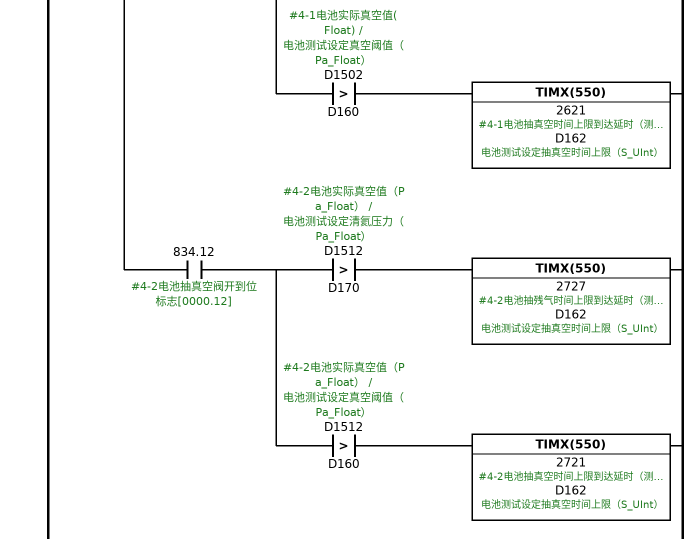
; [picture p648: Common / 动作延时, rungs 17-17]
; rung 17
LD P_On
OUT TR0
AND<=F(332) D1502 D160  ; #4-1电池实际真空值(Float), 电池测试设定真空阈值（Pa_Float）
LD 834.10  ; #4-1电池抽真空阀开到位标志[0000.10]
OR P_On
ANDLD
TIMX(550) 2620 #1  ; #4-1电池抽真空阈值到达延时（测试）
LD TR0
AND<=F(332) D1512 D160  ; #4-2电池实际真空值（Pa_Float）, 电池测试设定真空阈值（Pa_Float）
LD 834.12  ; #4-2电池抽真空阀开到位标志[0000.12]
OR P_On
ANDLD
TIMX(550) 2720 #1  ; #4-2电池抽真空阈值到达延时（测试）
LD TR0
LD>F(333) D1502 D172  ; #4-1电池实际真空值(Float), 电池测试设定破真空阈值（Pa_Float）
OR H5.15  ; 腔体模式（0-正压 1-负压）
ANDLD
TIMX(550) 2622 #1  ; #4-1电池破真空阈值到达延时（测试）
LD TR0
LD>F(333) D1512 D172  ; #4-2电池实际真空值（Pa_Float）, 电池测试设定破真空阈值（Pa_Float）
OR H5.15  ; 腔体模式（0-正压 1-负压）
ANDLD
TIMX(550) 2722 #1  ; #4-2电池破真空阈值到达延时（测试）
LD TR0
AND>=F(334) D1502 D176  ; #4-1电池实际真空值(Float), 电池测试设定注氦压力（Pa_Float）
AND 834.14  ; #4-1电池注氦阀开到位标志[0000.14]
TIMHX(551) 2624 #0  ; #4-1电池注氦压力到达延时（测试）
LD TR0
AND>=F(334) D1512 D176  ; #4-2电池实际真空值（Pa_Float）, 电池测试设定注氦压力（Pa_Float）
AND 835.00  ; #4-2电池注氦阀开到位标志[0000.00]
TIMHX(551) 2724 #0  ; #4-2电池注氦压力到达延时（测试）
LD TR0
AND<=F(332) D1502 D172  ; #4-1电池实际真空值(Float), 电池测试设定破真空阈值（Pa_Float）
AND 835.02  ; #4-1电池破真空阀开到位标志[0000.02]
TIMX(550) 2623 &20  ; #4-1电池破真空时间上限到达延时（测试）
LD TR0
AND<=F(332) D1512 D172  ; #4-2电池实际真空值（Pa_Float）, 电池测试设定破真空阈值（Pa_Float）
AND 835.04  ; #4-2电池破真空阀开到位标志[0000.04]
TIMX(550) 2723 &20  ; #4-2电池破真空时间上限到达延时（测试）
LD TR0
AND<=F(332) D1502 D170  ; #4-1电池实际真空值(Float), 电池测试设定清氦压力（Pa_Float）
TIMX(550) 2626 #1  ; #4-1电池抽残气压力到达延时（测试）
LD TR0
AND<=F(332) D1512 D170  ; #4-2电池实际真空值（Pa_Float）, 电池测试设定清氦压力（Pa_Float）
TIMX(550) 2726 #1  ; #4-2电池抽残气压力到达延时（测试）
LD TR0
AND>=F(334) D1502 D174  ; #4-1电池实际真空值(Float), 电池测试设定预抽检测压力（Pa_Float）
AND T2609  ; #4-1腔体预抽时间到达延时（测试）
TIMHX(551) 2628 #0  ; #4-1电池预抽压力正常判定延时（测试）
LD TR0
AND>=F(334) D1512 D174  ; #4-2电池实际真空值（Pa_Float）, 电池测试设定预抽检测压力（Pa_Float）
AND T2609  ; #4-1腔体预抽时间到达延时（测试）
TIMHX(551) 2728 #0  ; #4-2电池预抽压力正常判定延时（测试）
LD TR0
AND 834.14  ; #4-1电池注氦阀开到位标志[0000.14]
AND<F(331) D1502 D176  ; #4-1电池实际真空值(Float), 电池测试设定注氦压力（Pa_Float）
TIMX(550) 2625 D168  ; 电池测试设定注氦时间上限（S_UInt）, #4-1电池注氦时间上限到达延时（测试）
LD TR0
AND 835.00  ; #4-2电池注氦阀开到位标志[0000.00]
AND<F(331) D1512 D178  ; #4-2电池实际真空值（Pa_Float）, 注氦压力下限值（Pa_Float）
TIMX(550) 2725 D168  ; 电池测试设定注氦时间上限（S_UInt）, #4-2电池注氦时间上限到达延时（测试）
LD TR0
AND 834.10  ; #4-1电池抽真空阀开到位标志[0000.10]
OUT TR1
AND>F(333) D1502 D170  ; #4-1电池实际真空值(Float), 电池测试设定清氦压力（Pa_Float）
TIMX(550) 2627 D162  ; 电池测试设定抽真空时间上限（S_UInt）, #4-1电池抽残气时间上限到达延时（测试）
LD TR1
AND>F(333) D1502 D160  ; #4-1电池实际真空值(Float), 电池测试设定真空阈值（Pa_Float）
TIMX(550) 2621 D162  ; 电池测试设定抽真空时间上限（S_UInt）, #4-1电池抽真空时间上限到达延时（测试）
LD TR0
AND 834.12  ; #4-2电池抽真空阀开到位标志[0000.12]
OUT TR0
AND>F(333) D1512 D170  ; #4-2电池实际真空值（Pa_Float）, 电池测试设定清氦压力（Pa_Float）
TIMX(550) 2727 D162  ; 电池测试设定抽真空时间上限（S_UInt）, #4-2电池抽残气时间上限到达延时（测试）
LD TR0
AND>F(333) D1512 D160  ; #4-2电池实际真空值（Pa_Float）, 电池测试设定真空阈值（Pa_Float）
TIMX(550) 2721 D162  ; 电池测试设定抽真空时间上限（S_UInt）, #4-2电池抽真空时间上限到达延时（测试）

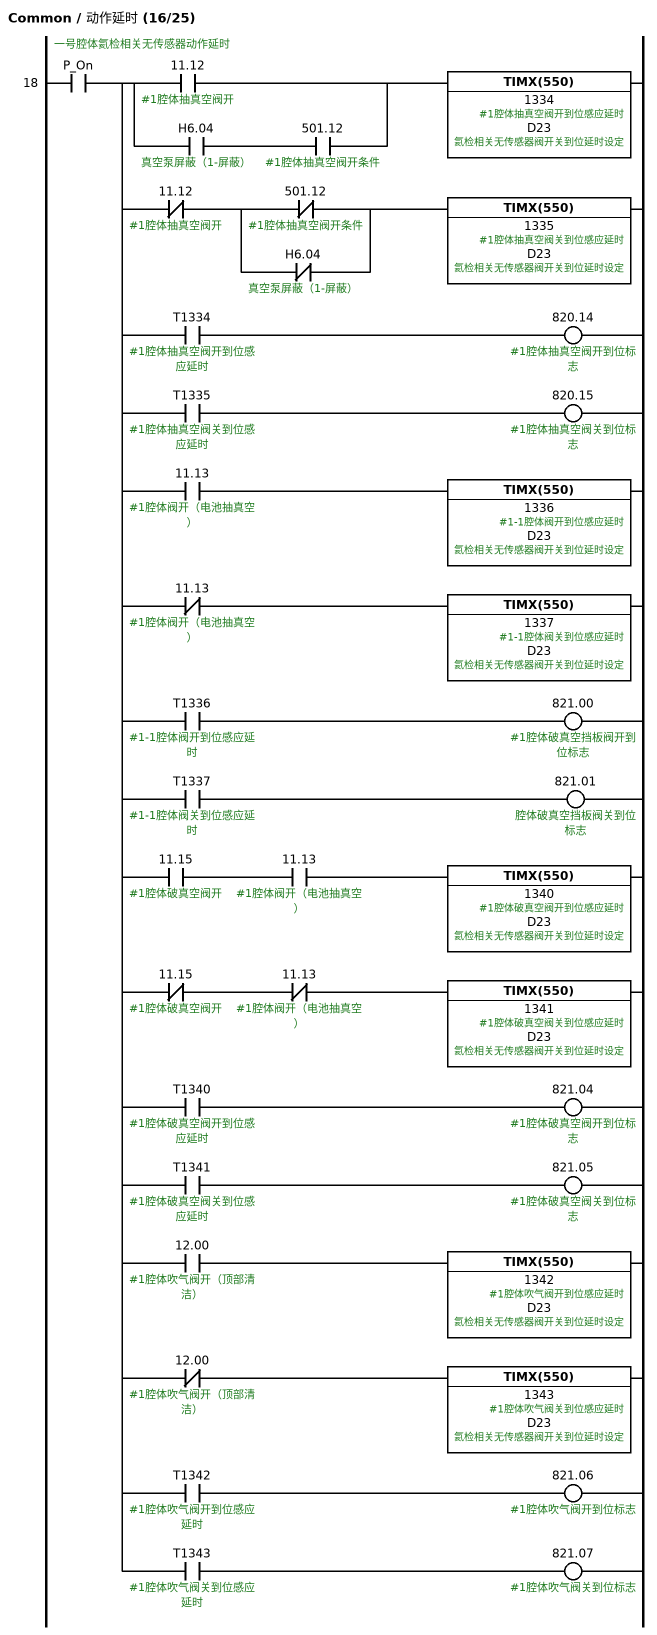
; rung 18: 一号腔体氦检相关无传感器动作延时
LD P_On
OUT TR0
LD 11.12  ; #1腔体抽真空阀开
LD H6.04  ; 真空泵屏蔽（1-屏蔽）
AND 501.12  ; #1腔体抽真空阀开条件
ORLD
ANDLD
TIMX(550) 1334 D23  ; 氦检相关无传感器阀开关到位延时设定, #1腔体抽真空阀开到位感应延时
LD TR0
ANDNOT 11.12  ; #1腔体抽真空阀开
LDNOT 501.12  ; #1腔体抽真空阀开条件
ORNOT H6.04  ; 真空泵屏蔽（1-屏蔽）
ANDLD
TIMX(550) 1335 D23  ; 氦检相关无传感器阀开关到位延时设定, #1腔体抽真空阀关到位感应延时
LD TR0
AND T1334  ; #1腔体抽真空阀开到位感应延时
OUT 820.14  ; #1腔体抽真空阀开到位标志
LD TR0
AND T1335  ; #1腔体抽真空阀关到位感应延时
OUT 820.15  ; #1腔体抽真空阀关到位标志
LD TR0
AND 11.13  ; #1腔体阀开（电池抽真空）
TIMX(550) 1336 D23  ; 氦检相关无传感器阀开关到位延时设定, #1-1腔体阀开到位感应延时
LD TR0
ANDNOT 11.13  ; #1腔体阀开（电池抽真空）
TIMX(550) 1337 D23  ; 氦检相关无传感器阀开关到位延时设定, #1-1腔体阀关到位感应延时
LD TR0
AND T1336  ; #1-1腔体阀开到位感应延时
OUT 821.00  ; #1腔体破真空挡板阀开到位标志
LD TR0
AND T1337  ; #1-1腔体阀关到位感应延时
OUT 821.01  ; 腔体破真空挡板阀关到位标志
LD TR0
AND 11.15  ; #1腔体破真空阀开
AND 11.13  ; #1腔体阀开（电池抽真空）
TIMX(550) 1340 D23  ; 氦检相关无传感器阀开关到位延时设定, #1腔体破真空阀开到位感应延时
LD TR0
ANDNOT 11.15  ; #1腔体破真空阀开
ANDNOT 11.13  ; #1腔体阀开（电池抽真空）
TIMX(550) 1341 D23  ; 氦检相关无传感器阀开关到位延时设定, #1腔体破真空阀关到位感应延时
LD TR0
AND T1340  ; #1腔体破真空阀开到位感应延时
OUT 821.04  ; #1腔体破真空阀开到位标志
LD TR0
AND T1341  ; #1腔体破真空阀关到位感应延时
OUT 821.05  ; #1腔体破真空阀关到位标志
LD TR0
AND 12.00  ; #1腔体吹气阀开（顶部清洁）
TIMX(550) 1342 D23  ; 氦检相关无传感器阀开关到位延时设定, #1腔体吹气阀开到位感应延时
LD TR0
ANDNOT 12.00  ; #1腔体吹气阀开（顶部清洁）
TIMX(550) 1343 D23  ; 氦检相关无传感器阀开关到位延时设定, #1腔体吹气阀关到位感应延时
LD TR0
AND T1342  ; #1腔体吹气阀开到位感应延时
OUT 821.06  ; #1腔体吹气阀开到位标志
LD TR0
AND T1343  ; #1腔体吹气阀关到位感应延时
OUT 821.07  ; #1腔体吹气阀关到位标志

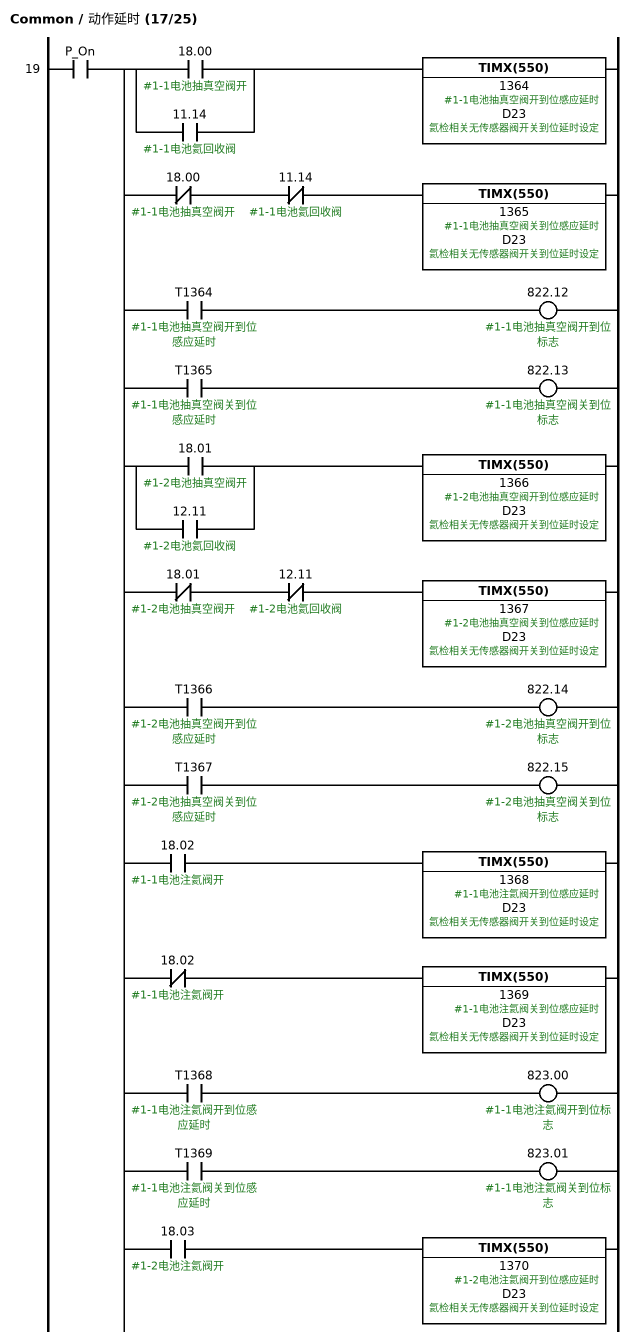

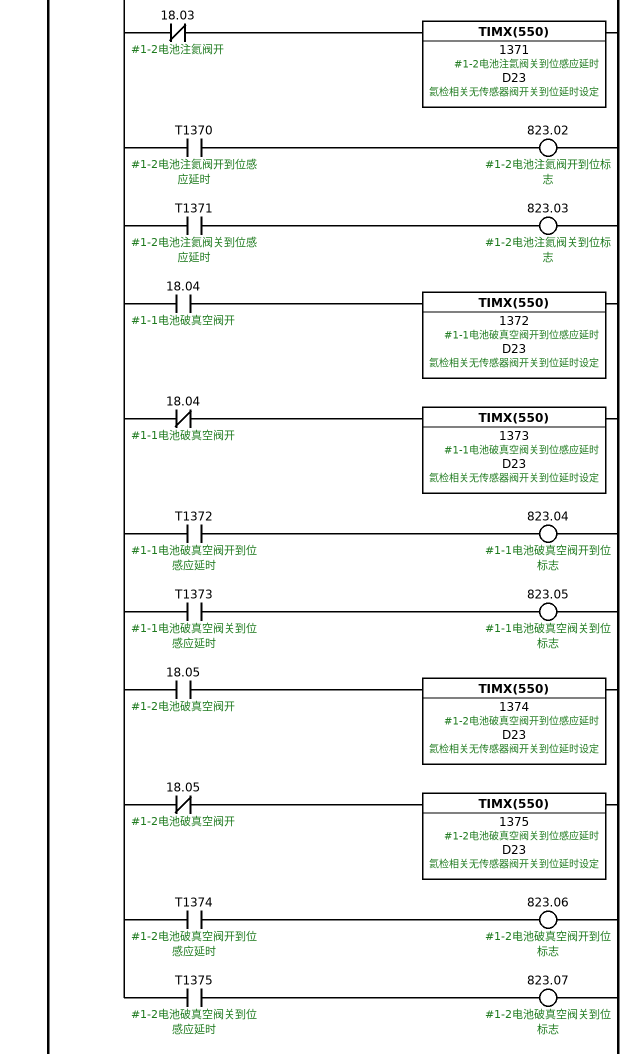
; rung 19
LD P_On
OUT TR0
LD 18.00  ; #1-1电池抽真空阀开
OR 11.14  ; #1-1电池氦回收阀
ANDLD
TIMX(550) 1364 D23  ; 氦检相关无传感器阀开关到位延时设定, #1-1电池抽真空阀开到位感应延时
LD TR0
ANDNOT 18.00  ; #1-1电池抽真空阀开
ANDNOT 11.14  ; #1-1电池氦回收阀
TIMX(550) 1365 D23  ; 氦检相关无传感器阀开关到位延时设定, #1-1电池抽真空阀关到位感应延时
LD TR0
AND T1364  ; #1-1电池抽真空阀开到位感应延时
OUT 822.12  ; #1-1电池抽真空阀开到位标志
LD TR0
AND T1365  ; #1-1电池抽真空阀关到位感应延时
OUT 822.13  ; #1-1电池抽真空阀关到位标志
LD TR0
LD 18.01  ; #1-2电池抽真空阀开
OR 12.11  ; #1-2电池氦回收阀
ANDLD
TIMX(550) 1366 D23  ; 氦检相关无传感器阀开关到位延时设定, #1-2电池抽真空阀开到位感应延时
LD TR0
ANDNOT 18.01  ; #1-2电池抽真空阀开
ANDNOT 12.11  ; #1-2电池氦回收阀
TIMX(550) 1367 D23  ; 氦检相关无传感器阀开关到位延时设定, #1-2电池抽真空阀关到位感应延时
LD TR0
AND T1366  ; #1-2电池抽真空阀开到位感应延时
OUT 822.14  ; #1-2电池抽真空阀开到位标志
LD TR0
AND T1367  ; #1-2电池抽真空阀关到位感应延时
OUT 822.15  ; #1-2电池抽真空阀关到位标志
LD TR0
AND 18.02  ; #1-1电池注氦阀开
TIMX(550) 1368 D23  ; 氦检相关无传感器阀开关到位延时设定, #1-1电池注氦阀开到位感应延时
LD TR0
ANDNOT 18.02  ; #1-1电池注氦阀开
TIMX(550) 1369 D23  ; 氦检相关无传感器阀开关到位延时设定, #1-1电池注氦阀关到位感应延时
LD TR0
AND T1368  ; #1-1电池注氦阀开到位感应延时
OUT 823.00  ; #1-1电池注氦阀开到位标志
LD TR0
AND T1369  ; #1-1电池注氦阀关到位感应延时
OUT 823.01  ; #1-1电池注氦阀关到位标志
LD TR0
AND 18.03  ; #1-2电池注氦阀开
TIMX(550) 1370 D23  ; 氦检相关无传感器阀开关到位延时设定, #1-2电池注氦阀开到位感应延时
LD TR0
ANDNOT 18.03  ; #1-2电池注氦阀开
TIMX(550) 1371 D23  ; 氦检相关无传感器阀开关到位延时设定, #1-2电池注氦阀关到位感应延时
LD TR0
AND T1370  ; #1-2电池注氦阀开到位感应延时
OUT 823.02  ; #1-2电池注氦阀开到位标志
LD TR0
AND T1371  ; #1-2电池注氦阀关到位感应延时
OUT 823.03  ; #1-2电池注氦阀关到位标志
LD TR0
AND 18.04  ; #1-1电池破真空阀开
TIMX(550) 1372 D23  ; 氦检相关无传感器阀开关到位延时设定, #1-1电池破真空阀开到位感应延时
LD TR0
ANDNOT 18.04  ; #1-1电池破真空阀开
TIMX(550) 1373 D23  ; 氦检相关无传感器阀开关到位延时设定, #1-1电池破真空阀关到位感应延时
LD TR0
AND T1372  ; #1-1电池破真空阀开到位感应延时
OUT 823.04  ; #1-1电池破真空阀开到位标志
LD TR0
AND T1373  ; #1-1电池破真空阀关到位感应延时
OUT 823.05  ; #1-1电池破真空阀关到位标志
LD TR0
AND 18.05  ; #1-2电池破真空阀开
TIMX(550) 1374 D23  ; 氦检相关无传感器阀开关到位延时设定, #1-2电池破真空阀开到位感应延时
LD TR0
ANDNOT 18.05  ; #1-2电池破真空阀开
TIMX(550) 1375 D23  ; 氦检相关无传感器阀开关到位延时设定, #1-2电池破真空阀关到位感应延时
LD TR0
AND T1374  ; #1-2电池破真空阀开到位感应延时
OUT 823.06  ; #1-2电池破真空阀开到位标志
LD TR0
AND T1375  ; #1-2电池破真空阀关到位感应延时
OUT 823.07  ; #1-2电池破真空阀关到位标志

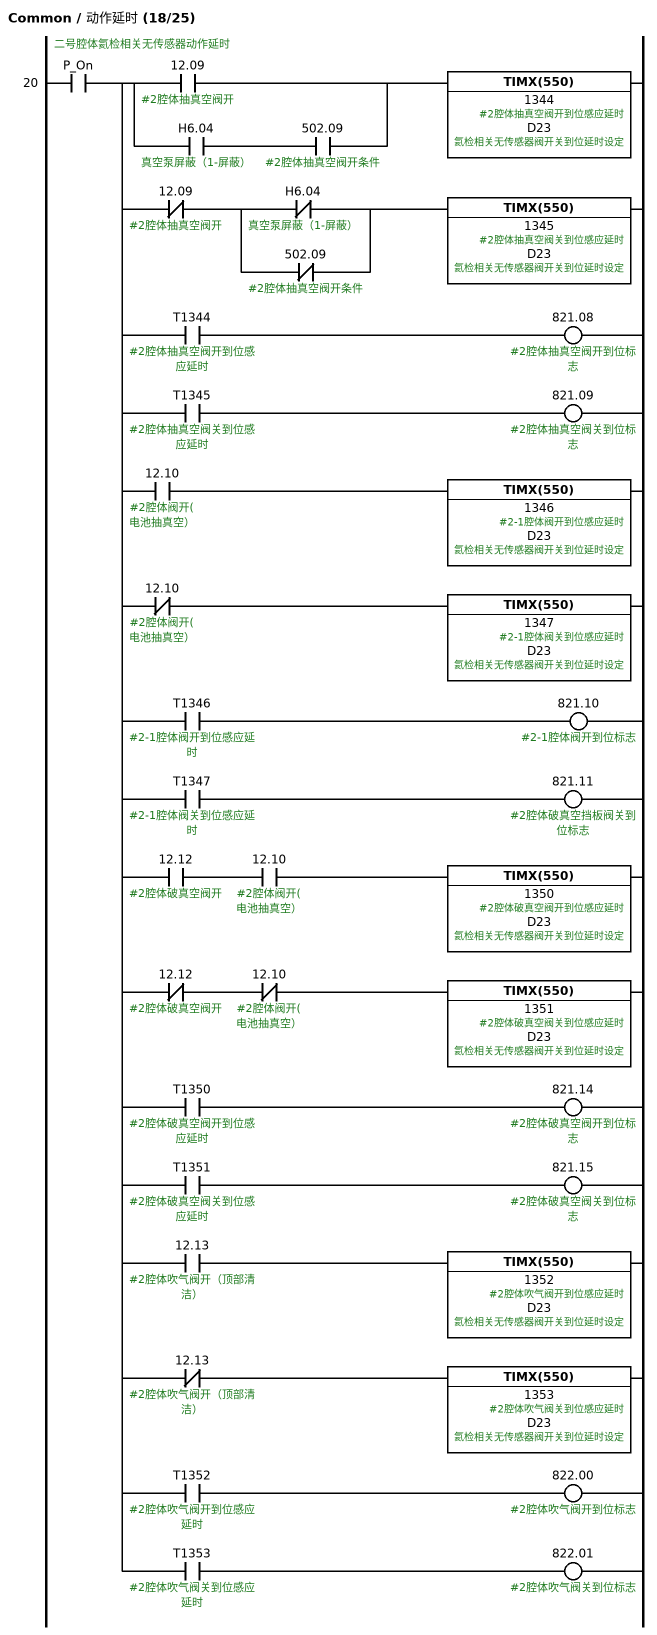
; rung 20: 二号腔体氦检相关无传感器动作延时
LD P_On
OUT TR0
LD 12.09  ; #2腔体抽真空阀开
LD H6.04  ; 真空泵屏蔽（1-屏蔽）
AND 502.09  ; #2腔体抽真空阀开条件
ORLD
ANDLD
TIMX(550) 1344 D23  ; 氦检相关无传感器阀开关到位延时设定, #2腔体抽真空阀开到位感应延时
LD TR0
ANDNOT 12.09  ; #2腔体抽真空阀开
LDNOT H6.04  ; 真空泵屏蔽（1-屏蔽）
ORNOT 502.09  ; #2腔体抽真空阀开条件
ANDLD
TIMX(550) 1345 D23  ; 氦检相关无传感器阀开关到位延时设定, #2腔体抽真空阀关到位感应延时
LD TR0
AND T1344  ; #2腔体抽真空阀开到位感应延时
OUT 821.08  ; #2腔体抽真空阀开到位标志
LD TR0
AND T1345  ; #2腔体抽真空阀关到位感应延时
OUT 821.09  ; #2腔体抽真空阀关到位标志
LD TR0
AND 12.10  ; #2腔体阀开(电池抽真空）
TIMX(550) 1346 D23  ; 氦检相关无传感器阀开关到位延时设定, #2-1腔体阀开到位感应延时
LD TR0
ANDNOT 12.10  ; #2腔体阀开(电池抽真空）
TIMX(550) 1347 D23  ; 氦检相关无传感器阀开关到位延时设定, #2-1腔体阀关到位感应延时
LD TR0
AND T1346  ; #2-1腔体阀开到位感应延时
OUT 821.10  ; #2-1腔体阀开到位标志
LD TR0
AND T1347  ; #2-1腔体阀关到位感应延时
OUT 821.11  ; #2腔体破真空挡板阀关到位标志
LD TR0
AND 12.12  ; #2腔体破真空阀开
AND 12.10  ; #2腔体阀开(电池抽真空）
TIMX(550) 1350 D23  ; 氦检相关无传感器阀开关到位延时设定, #2腔体破真空阀开到位感应延时
LD TR0
ANDNOT 12.12  ; #2腔体破真空阀开
ANDNOT 12.10  ; #2腔体阀开(电池抽真空）
TIMX(550) 1351 D23  ; 氦检相关无传感器阀开关到位延时设定, #2腔体破真空阀关到位感应延时
LD TR0
AND T1350  ; #2腔体破真空阀开到位感应延时
OUT 821.14  ; #2腔体破真空阀开到位标志
LD TR0
AND T1351  ; #2腔体破真空阀关到位感应延时
OUT 821.15  ; #2腔体破真空阀关到位标志
LD TR0
AND 12.13  ; #2腔体吹气阀开（顶部清洁）
TIMX(550) 1352 D23  ; 氦检相关无传感器阀开关到位延时设定, #2腔体吹气阀开到位感应延时
LD TR0
ANDNOT 12.13  ; #2腔体吹气阀开（顶部清洁）
TIMX(550) 1353 D23  ; 氦检相关无传感器阀开关到位延时设定, #2腔体吹气阀关到位感应延时
LD TR0
AND T1352  ; #2腔体吹气阀开到位感应延时
OUT 822.00  ; #2腔体吹气阀开到位标志
LD TR0
AND T1353  ; #2腔体吹气阀关到位感应延时
OUT 822.01  ; #2腔体吹气阀关到位标志

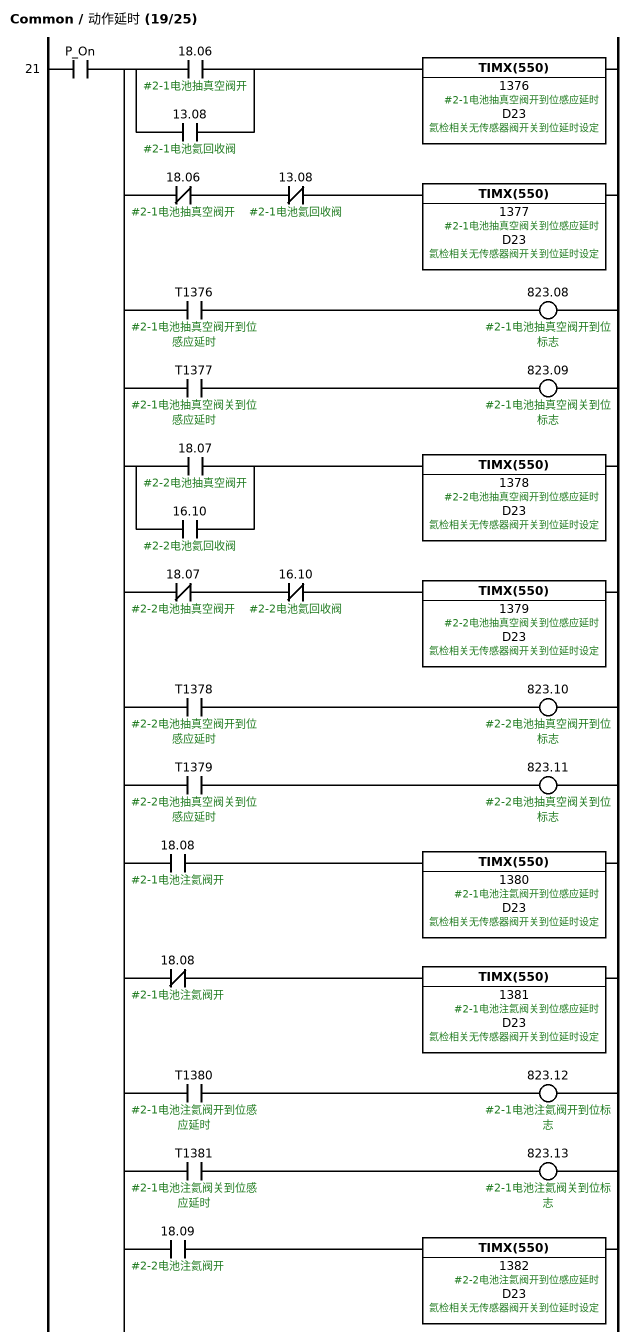

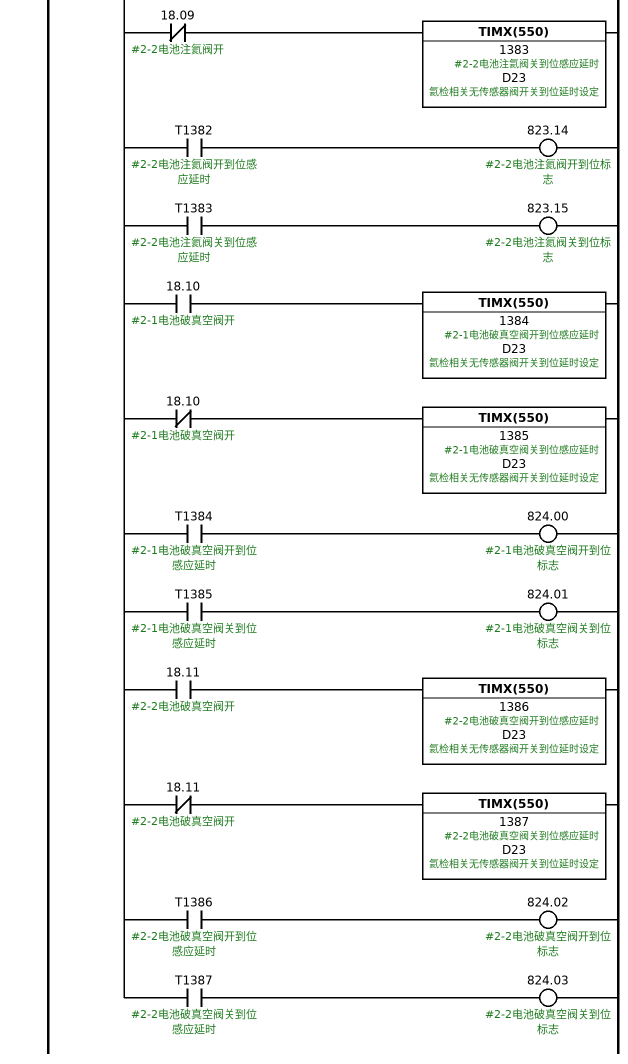
; rung 21
LD P_On
OUT TR0
LD 18.06  ; #2-1电池抽真空阀开
OR 13.08  ; #2-1电池氦回收阀
ANDLD
TIMX(550) 1376 D23  ; 氦检相关无传感器阀开关到位延时设定, #2-1电池抽真空阀开到位感应延时
LD TR0
ANDNOT 18.06  ; #2-1电池抽真空阀开
ANDNOT 13.08  ; #2-1电池氦回收阀
TIMX(550) 1377 D23  ; 氦检相关无传感器阀开关到位延时设定, #2-1电池抽真空阀关到位感应延时
LD TR0
AND T1376  ; #2-1电池抽真空阀开到位感应延时
OUT 823.08  ; #2-1电池抽真空阀开到位标志
LD TR0
AND T1377  ; #2-1电池抽真空阀关到位感应延时
OUT 823.09  ; #2-1电池抽真空阀关到位标志
LD TR0
LD 18.07  ; #2-2电池抽真空阀开
OR 16.10  ; #2-2电池氦回收阀
ANDLD
TIMX(550) 1378 D23  ; 氦检相关无传感器阀开关到位延时设定, #2-2电池抽真空阀开到位感应延时
LD TR0
ANDNOT 18.07  ; #2-2电池抽真空阀开
ANDNOT 16.10  ; #2-2电池氦回收阀
TIMX(550) 1379 D23  ; 氦检相关无传感器阀开关到位延时设定, #2-2电池抽真空阀关到位感应延时
LD TR0
AND T1378  ; #2-2电池抽真空阀开到位感应延时
OUT 823.10  ; #2-2电池抽真空阀开到位标志
LD TR0
AND T1379  ; #2-2电池抽真空阀关到位感应延时
OUT 823.11  ; #2-2电池抽真空阀关到位标志
LD TR0
AND 18.08  ; #2-1电池注氦阀开
TIMX(550) 1380 D23  ; 氦检相关无传感器阀开关到位延时设定, #2-1电池注氦阀开到位感应延时
LD TR0
ANDNOT 18.08  ; #2-1电池注氦阀开
TIMX(550) 1381 D23  ; 氦检相关无传感器阀开关到位延时设定, #2-1电池注氦阀关到位感应延时
LD TR0
AND T1380  ; #2-1电池注氦阀开到位感应延时
OUT 823.12  ; #2-1电池注氦阀开到位标志
LD TR0
AND T1381  ; #2-1电池注氦阀关到位感应延时
OUT 823.13  ; #2-1电池注氦阀关到位标志
LD TR0
AND 18.09  ; #2-2电池注氦阀开
TIMX(550) 1382 D23  ; 氦检相关无传感器阀开关到位延时设定, #2-2电池注氦阀开到位感应延时
LD TR0
ANDNOT 18.09  ; #2-2电池注氦阀开
TIMX(550) 1383 D23  ; 氦检相关无传感器阀开关到位延时设定, #2-2电池注氦阀关到位感应延时
LD TR0
AND T1382  ; #2-2电池注氦阀开到位感应延时
OUT 823.14  ; #2-2电池注氦阀开到位标志
LD TR0
AND T1383  ; #2-2电池注氦阀关到位感应延时
OUT 823.15  ; #2-2电池注氦阀关到位标志
LD TR0
AND 18.10  ; #2-1电池破真空阀开
TIMX(550) 1384 D23  ; 氦检相关无传感器阀开关到位延时设定, #2-1电池破真空阀开到位感应延时
LD TR0
ANDNOT 18.10  ; #2-1电池破真空阀开
TIMX(550) 1385 D23  ; 氦检相关无传感器阀开关到位延时设定, #2-1电池破真空阀关到位感应延时
LD TR0
AND T1384  ; #2-1电池破真空阀开到位感应延时
OUT 824.00  ; #2-1电池破真空阀开到位标志
LD TR0
AND T1385  ; #2-1电池破真空阀关到位感应延时
OUT 824.01  ; #2-1电池破真空阀关到位标志
LD TR0
AND 18.11  ; #2-2电池破真空阀开
TIMX(550) 1386 D23  ; 氦检相关无传感器阀开关到位延时设定, #2-2电池破真空阀开到位感应延时
LD TR0
ANDNOT 18.11  ; #2-2电池破真空阀开
TIMX(550) 1387 D23  ; 氦检相关无传感器阀开关到位延时设定, #2-2电池破真空阀关到位感应延时
LD TR0
AND T1386  ; #2-2电池破真空阀开到位感应延时
OUT 824.02  ; #2-2电池破真空阀开到位标志
LD TR0
AND T1387  ; #2-2电池破真空阀关到位感应延时
OUT 824.03  ; #2-2电池破真空阀关到位标志

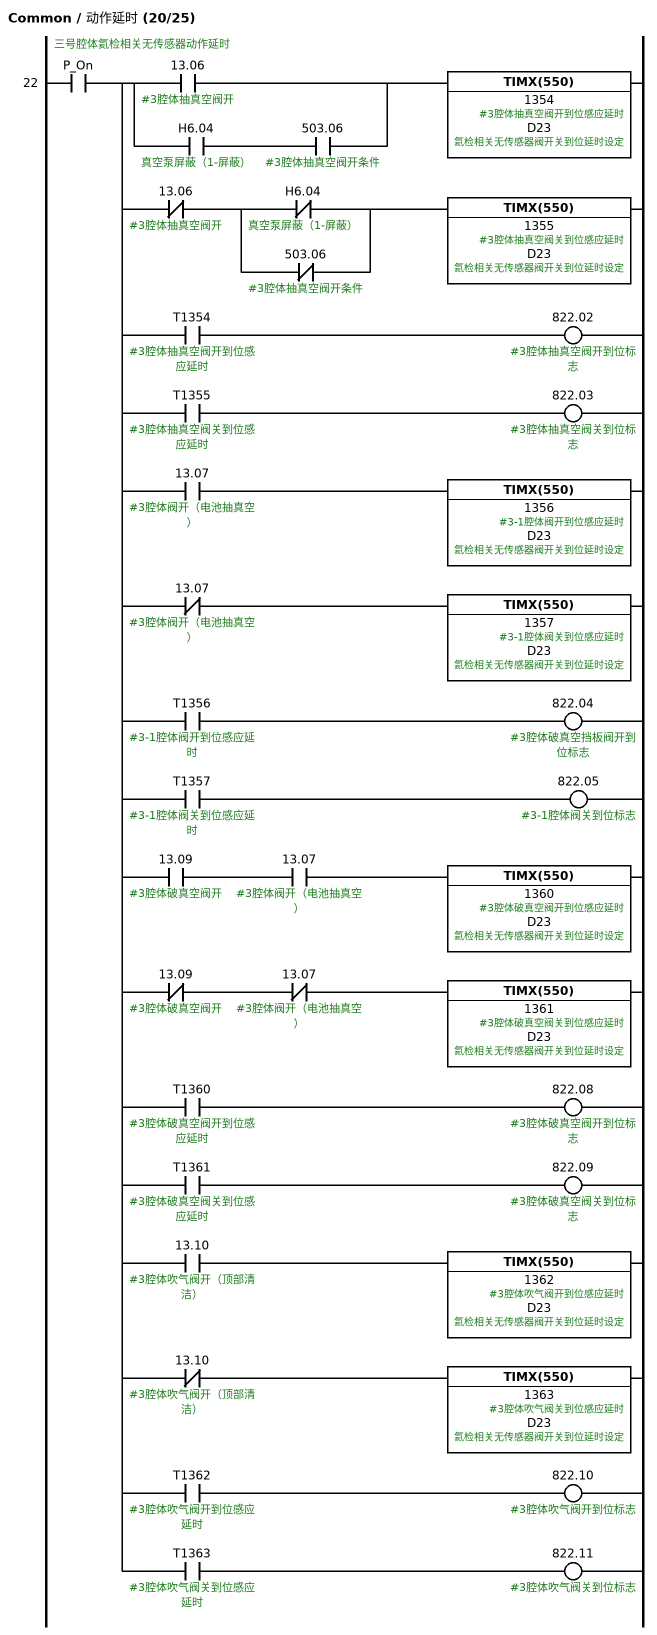
; rung 22: 三号腔体氦检相关无传感器动作延时
LD P_On
OUT TR0
LD 13.06  ; #3腔体抽真空阀开
LD H6.04  ; 真空泵屏蔽（1-屏蔽）
AND 503.06  ; #3腔体抽真空阀开条件
ORLD
ANDLD
TIMX(550) 1354 D23  ; 氦检相关无传感器阀开关到位延时设定, #3腔体抽真空阀开到位感应延时
LD TR0
ANDNOT 13.06  ; #3腔体抽真空阀开
LDNOT H6.04  ; 真空泵屏蔽（1-屏蔽）
ORNOT 503.06  ; #3腔体抽真空阀开条件
ANDLD
TIMX(550) 1355 D23  ; 氦检相关无传感器阀开关到位延时设定, #3腔体抽真空阀关到位感应延时
LD TR0
AND T1354  ; #3腔体抽真空阀开到位感应延时
OUT 822.02  ; #3腔体抽真空阀开到位标志
LD TR0
AND T1355  ; #3腔体抽真空阀关到位感应延时
OUT 822.03  ; #3腔体抽真空阀关到位标志
LD TR0
AND 13.07  ; #3腔体阀开（电池抽真空）
TIMX(550) 1356 D23  ; 氦检相关无传感器阀开关到位延时设定, #3-1腔体阀开到位感应延时
LD TR0
ANDNOT 13.07  ; #3腔体阀开（电池抽真空）
TIMX(550) 1357 D23  ; 氦检相关无传感器阀开关到位延时设定, #3-1腔体阀关到位感应延时
LD TR0
AND T1356  ; #3-1腔体阀开到位感应延时
OUT 822.04  ; #3腔体破真空挡板阀开到位标志
LD TR0
AND T1357  ; #3-1腔体阀关到位感应延时
OUT 822.05  ; #3-1腔体阀关到位标志
LD TR0
AND 13.09  ; #3腔体破真空阀开
AND 13.07  ; #3腔体阀开（电池抽真空）
TIMX(550) 1360 D23  ; 氦检相关无传感器阀开关到位延时设定, #3腔体破真空阀开到位感应延时
LD TR0
ANDNOT 13.09  ; #3腔体破真空阀开
ANDNOT 13.07  ; #3腔体阀开（电池抽真空）
TIMX(550) 1361 D23  ; 氦检相关无传感器阀开关到位延时设定, #3腔体破真空阀关到位感应延时
LD TR0
AND T1360  ; #3腔体破真空阀开到位感应延时
OUT 822.08  ; #3腔体破真空阀开到位标志
LD TR0
AND T1361  ; #3腔体破真空阀关到位感应延时
OUT 822.09  ; #3腔体破真空阀关到位标志
LD TR0
AND 13.10  ; #3腔体吹气阀开（顶部清洁）
TIMX(550) 1362 D23  ; 氦检相关无传感器阀开关到位延时设定, #3腔体吹气阀开到位感应延时
LD TR0
ANDNOT 13.10  ; #3腔体吹气阀开（顶部清洁）
TIMX(550) 1363 D23  ; 氦检相关无传感器阀开关到位延时设定, #3腔体吹气阀关到位感应延时
LD TR0
AND T1362  ; #3腔体吹气阀开到位感应延时
OUT 822.10  ; #3腔体吹气阀开到位标志
LD TR0
AND T1363  ; #3腔体吹气阀关到位感应延时
OUT 822.11  ; #3腔体吹气阀关到位标志

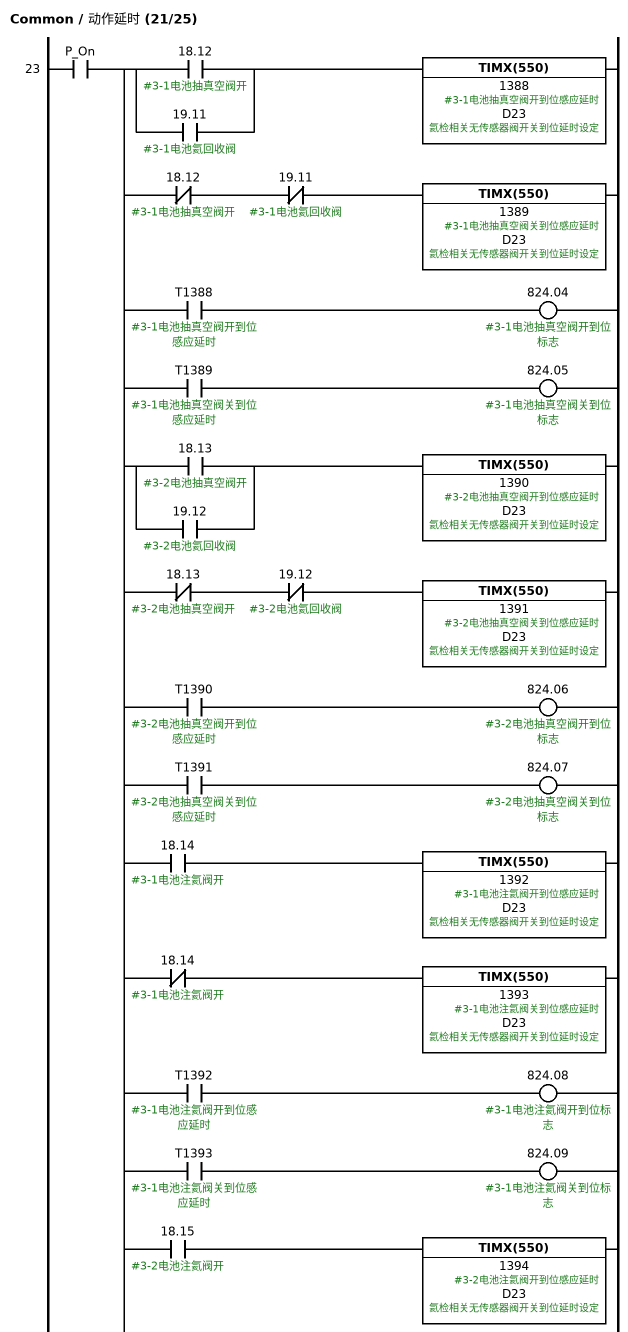

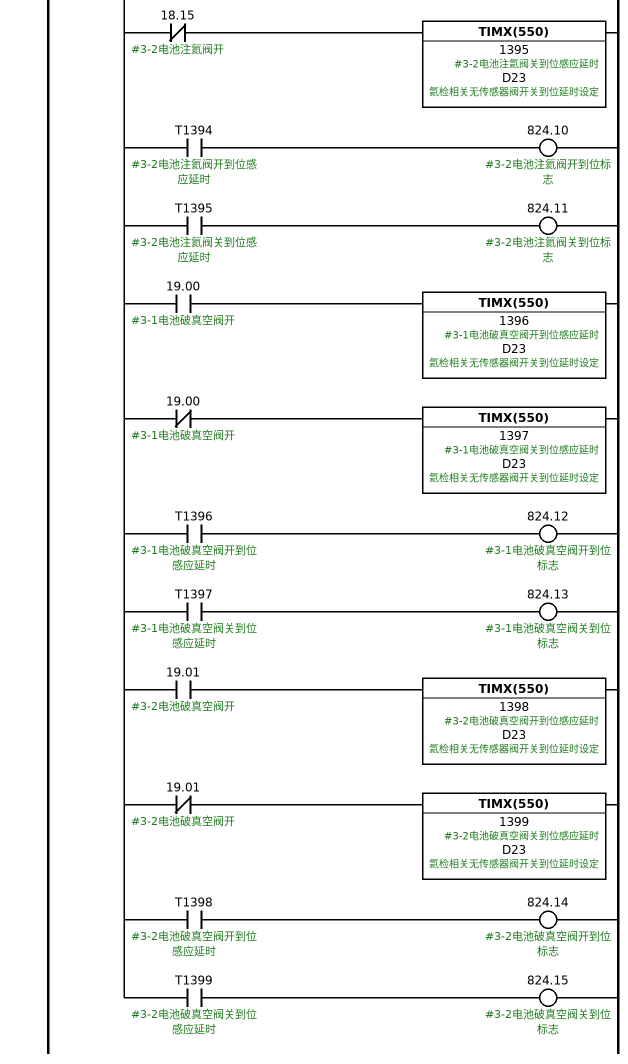
; rung 23
LD P_On
OUT TR0
LD 18.12  ; #3-1电池抽真空阀开
OR 19.11  ; #3-1电池氦回收阀
ANDLD
TIMX(550) 1388 D23  ; 氦检相关无传感器阀开关到位延时设定, #3-1电池抽真空阀开到位感应延时
LD TR0
ANDNOT 18.12  ; #3-1电池抽真空阀开
ANDNOT 19.11  ; #3-1电池氦回收阀
TIMX(550) 1389 D23  ; 氦检相关无传感器阀开关到位延时设定, #3-1电池抽真空阀关到位感应延时
LD TR0
AND T1388  ; #3-1电池抽真空阀开到位感应延时
OUT 824.04  ; #3-1电池抽真空阀开到位标志
LD TR0
AND T1389  ; #3-1电池抽真空阀关到位感应延时
OUT 824.05  ; #3-1电池抽真空阀关到位标志
LD TR0
LD 18.13  ; #3-2电池抽真空阀开
OR 19.12  ; #3-2电池氦回收阀
ANDLD
TIMX(550) 1390 D23  ; 氦检相关无传感器阀开关到位延时设定, #3-2电池抽真空阀开到位感应延时
LD TR0
ANDNOT 18.13  ; #3-2电池抽真空阀开
ANDNOT 19.12  ; #3-2电池氦回收阀
TIMX(550) 1391 D23  ; 氦检相关无传感器阀开关到位延时设定, #3-2电池抽真空阀关到位感应延时
LD TR0
AND T1390  ; #3-2电池抽真空阀开到位感应延时
OUT 824.06  ; #3-2电池抽真空阀开到位标志
LD TR0
AND T1391  ; #3-2电池抽真空阀关到位感应延时
OUT 824.07  ; #3-2电池抽真空阀关到位标志
LD TR0
AND 18.14  ; #3-1电池注氦阀开
TIMX(550) 1392 D23  ; 氦检相关无传感器阀开关到位延时设定, #3-1电池注氦阀开到位感应延时
LD TR0
ANDNOT 18.14  ; #3-1电池注氦阀开
TIMX(550) 1393 D23  ; 氦检相关无传感器阀开关到位延时设定, #3-1电池注氦阀关到位感应延时
LD TR0
AND T1392  ; #3-1电池注氦阀开到位感应延时
OUT 824.08  ; #3-1电池注氦阀开到位标志
LD TR0
AND T1393  ; #3-1电池注氦阀关到位感应延时
OUT 824.09  ; #3-1电池注氦阀关到位标志
LD TR0
AND 18.15  ; #3-2电池注氦阀开
TIMX(550) 1394 D23  ; 氦检相关无传感器阀开关到位延时设定, #3-2电池注氦阀开到位感应延时
LD TR0
ANDNOT 18.15  ; #3-2电池注氦阀开
TIMX(550) 1395 D23  ; 氦检相关无传感器阀开关到位延时设定, #3-2电池注氦阀关到位感应延时
LD TR0
AND T1394  ; #3-2电池注氦阀开到位感应延时
OUT 824.10  ; #3-2电池注氦阀开到位标志
LD TR0
AND T1395  ; #3-2电池注氦阀关到位感应延时
OUT 824.11  ; #3-2电池注氦阀关到位标志
LD TR0
AND 19.00  ; #3-1电池破真空阀开
TIMX(550) 1396 D23  ; 氦检相关无传感器阀开关到位延时设定, #3-1电池破真空阀开到位感应延时
LD TR0
ANDNOT 19.00  ; #3-1电池破真空阀开
TIMX(550) 1397 D23  ; 氦检相关无传感器阀开关到位延时设定, #3-1电池破真空阀关到位感应延时
LD TR0
AND T1396  ; #3-1电池破真空阀开到位感应延时
OUT 824.12  ; #3-1电池破真空阀开到位标志
LD TR0
AND T1397  ; #3-1电池破真空阀关到位感应延时
OUT 824.13  ; #3-1电池破真空阀关到位标志
LD TR0
AND 19.01  ; #3-2电池破真空阀开
TIMX(550) 1398 D23  ; 氦检相关无传感器阀开关到位延时设定, #3-2电池破真空阀开到位感应延时
LD TR0
ANDNOT 19.01  ; #3-2电池破真空阀开
TIMX(550) 1399 D23  ; 氦检相关无传感器阀开关到位延时设定, #3-2电池破真空阀关到位感应延时
LD TR0
AND T1398  ; #3-2电池破真空阀开到位感应延时
OUT 824.14  ; #3-2电池破真空阀开到位标志
LD TR0
AND T1399  ; #3-2电池破真空阀关到位感应延时
OUT 824.15  ; #3-2电池破真空阀关到位标志

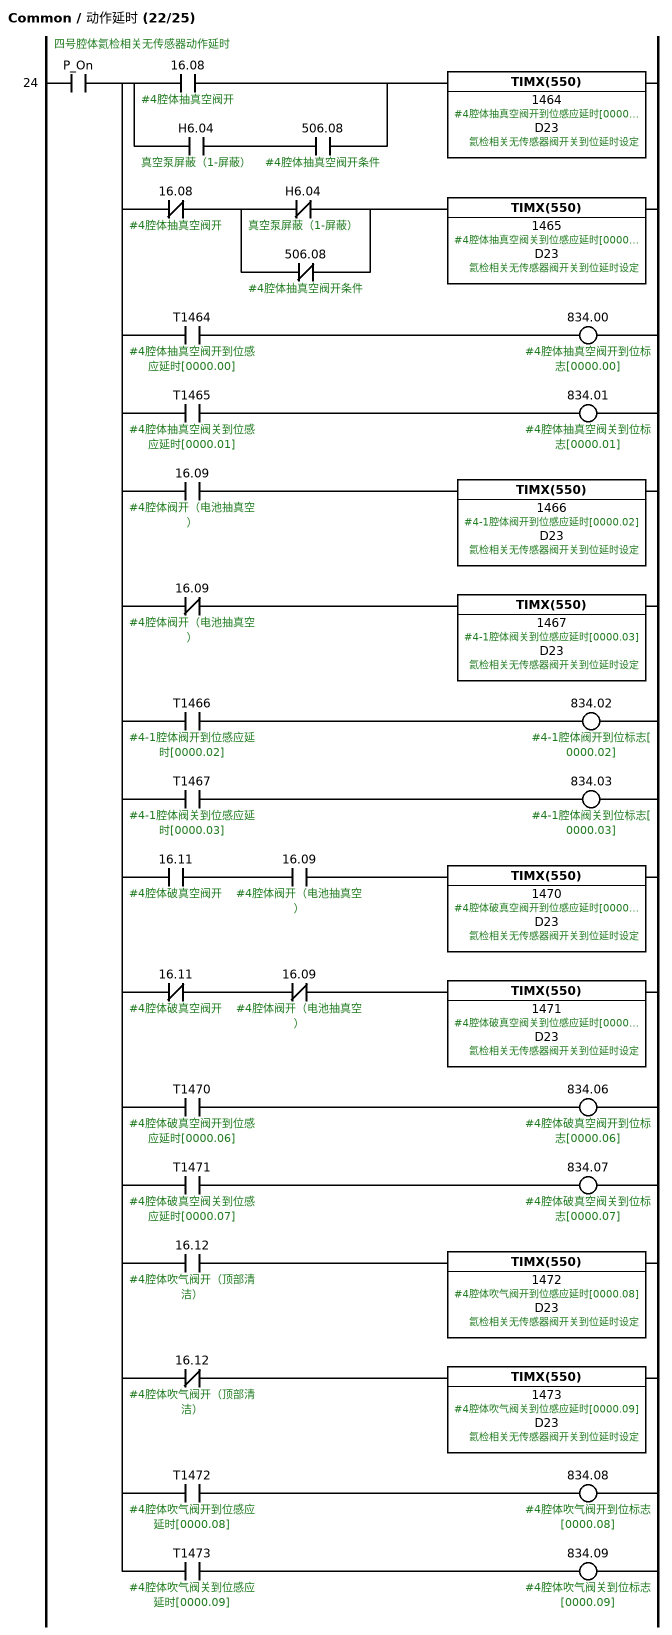
; rung 24: 四号腔体氦检相关无传感器动作延时
LD P_On
OUT TR0
LD 16.08  ; #4腔体抽真空阀开
LD H6.04  ; 真空泵屏蔽（1-屏蔽）
AND 506.08  ; #4腔体抽真空阀开条件
ORLD
ANDLD
TIMX(550) 1464 D23  ; 氦检相关无传感器阀开关到位延时设定, #4腔体抽真空阀开到位感应延时[0000.00]
LD TR0
ANDNOT 16.08  ; #4腔体抽真空阀开
LDNOT H6.04  ; 真空泵屏蔽（1-屏蔽）
ORNOT 506.08  ; #4腔体抽真空阀开条件
ANDLD
TIMX(550) 1465 D23  ; 氦检相关无传感器阀开关到位延时设定, #4腔体抽真空阀关到位感应延时[0000.01]
LD TR0
AND T1464  ; #4腔体抽真空阀开到位感应延时[0000.00]
OUT 834.00  ; #4腔体抽真空阀开到位标志[0000.00]
LD TR0
AND T1465  ; #4腔体抽真空阀关到位感应延时[0000.01]
OUT 834.01  ; #4腔体抽真空阀关到位标志[0000.01]
LD TR0
AND 16.09  ; #4腔体阀开（电池抽真空）
TIMX(550) 1466 D23  ; 氦检相关无传感器阀开关到位延时设定, #4-1腔体阀开到位感应延时[0000.02]
LD TR0
ANDNOT 16.09  ; #4腔体阀开（电池抽真空）
TIMX(550) 1467 D23  ; 氦检相关无传感器阀开关到位延时设定, #4-1腔体阀关到位感应延时[0000.03]
LD TR0
AND T1466  ; #4-1腔体阀开到位感应延时[0000.02]
OUT 834.02  ; #4-1腔体阀开到位标志[0000.02]
LD TR0
AND T1467  ; #4-1腔体阀关到位感应延时[0000.03]
OUT 834.03  ; #4-1腔体阀关到位标志[0000.03]
LD TR0
AND 16.11  ; #4腔体破真空阀开
AND 16.09  ; #4腔体阀开（电池抽真空）
TIMX(550) 1470 D23  ; 氦检相关无传感器阀开关到位延时设定, #4腔体破真空阀开到位感应延时[0000.06]
LD TR0
ANDNOT 16.11  ; #4腔体破真空阀开
ANDNOT 16.09  ; #4腔体阀开（电池抽真空）
TIMX(550) 1471 D23  ; 氦检相关无传感器阀开关到位延时设定, #4腔体破真空阀关到位感应延时[0000.07]
LD TR0
AND T1470  ; #4腔体破真空阀开到位感应延时[0000.06]
OUT 834.06  ; #4腔体破真空阀开到位标志[0000.06]
LD TR0
AND T1471  ; #4腔体破真空阀关到位感应延时[0000.07]
OUT 834.07  ; #4腔体破真空阀关到位标志[0000.07]
LD TR0
AND 16.12  ; #4腔体吹气阀开（顶部清洁）
TIMX(550) 1472 D23  ; 氦检相关无传感器阀开关到位延时设定, #4腔体吹气阀开到位感应延时[0000.08]
LD TR0
ANDNOT 16.12  ; #4腔体吹气阀开（顶部清洁）
TIMX(550) 1473 D23  ; 氦检相关无传感器阀开关到位延时设定, #4腔体吹气阀关到位感应延时[0000.09]
LD TR0
AND T1472  ; #4腔体吹气阀开到位感应延时[0000.08]
OUT 834.08  ; #4腔体吹气阀开到位标志[0000.08]
LD TR0
AND T1473  ; #4腔体吹气阀关到位感应延时[0000.09]
OUT 834.09  ; #4腔体吹气阀关到位标志[0000.09]

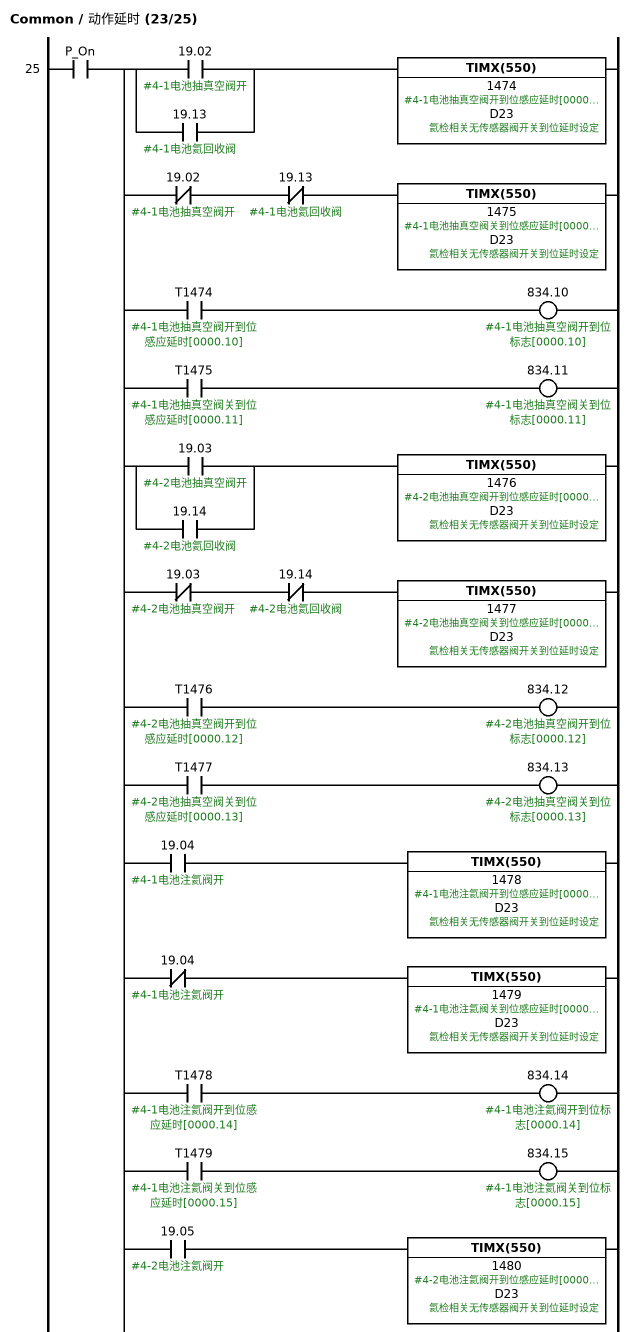

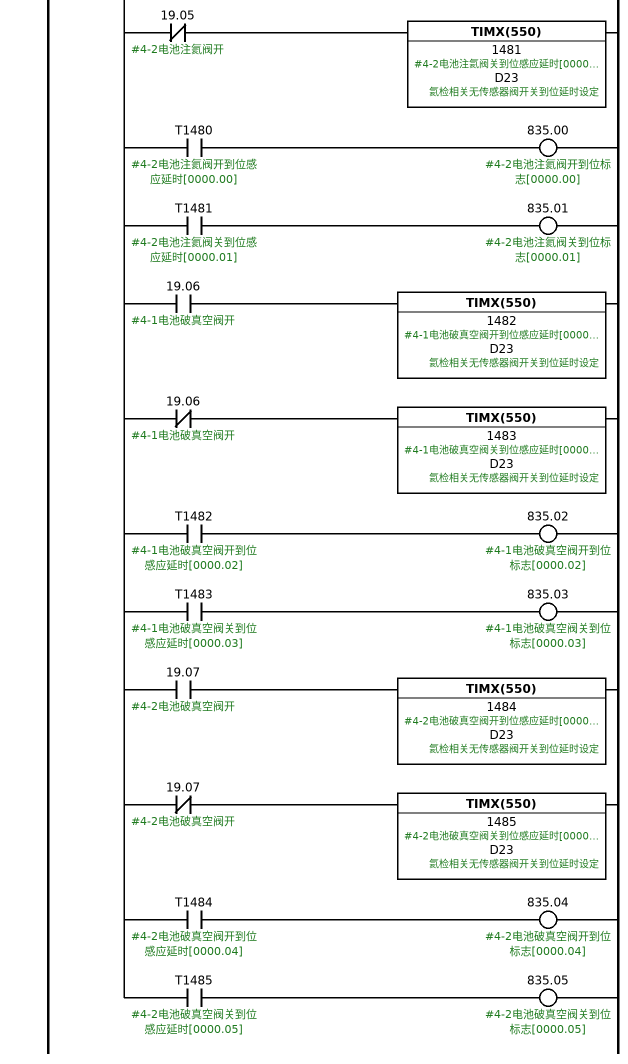
; rung 25
LD P_On
OUT TR0
LD 19.02  ; #4-1电池抽真空阀开
OR 19.13  ; #4-1电池氦回收阀
ANDLD
TIMX(550) 1474 D23  ; 氦检相关无传感器阀开关到位延时设定, #4-1电池抽真空阀开到位感应延时[0000.10]
LD TR0
ANDNOT 19.02  ; #4-1电池抽真空阀开
ANDNOT 19.13  ; #4-1电池氦回收阀
TIMX(550) 1475 D23  ; 氦检相关无传感器阀开关到位延时设定, #4-1电池抽真空阀关到位感应延时[0000.11]
LD TR0
AND T1474  ; #4-1电池抽真空阀开到位感应延时[0000.10]
OUT 834.10  ; #4-1电池抽真空阀开到位标志[0000.10]
LD TR0
AND T1475  ; #4-1电池抽真空阀关到位感应延时[0000.11]
OUT 834.11  ; #4-1电池抽真空阀关到位标志[0000.11]
LD TR0
LD 19.03  ; #4-2电池抽真空阀开
OR 19.14  ; #4-2电池氦回收阀
ANDLD
TIMX(550) 1476 D23  ; 氦检相关无传感器阀开关到位延时设定, #4-2电池抽真空阀开到位感应延时[0000.12]
LD TR0
ANDNOT 19.03  ; #4-2电池抽真空阀开
ANDNOT 19.14  ; #4-2电池氦回收阀
TIMX(550) 1477 D23  ; 氦检相关无传感器阀开关到位延时设定, #4-2电池抽真空阀关到位感应延时[0000.13]
LD TR0
AND T1476  ; #4-2电池抽真空阀开到位感应延时[0000.12]
OUT 834.12  ; #4-2电池抽真空阀开到位标志[0000.12]
LD TR0
AND T1477  ; #4-2电池抽真空阀关到位感应延时[0000.13]
OUT 834.13  ; #4-2电池抽真空阀关到位标志[0000.13]
LD TR0
AND 19.04  ; #4-1电池注氦阀开
TIMX(550) 1478 D23  ; 氦检相关无传感器阀开关到位延时设定, #4-1电池注氦阀开到位感应延时[0000.14]
LD TR0
ANDNOT 19.04  ; #4-1电池注氦阀开
TIMX(550) 1479 D23  ; 氦检相关无传感器阀开关到位延时设定, #4-1电池注氦阀关到位感应延时[0000.15]
LD TR0
AND T1478  ; #4-1电池注氦阀开到位感应延时[0000.14]
OUT 834.14  ; #4-1电池注氦阀开到位标志[0000.14]
LD TR0
AND T1479  ; #4-1电池注氦阀关到位感应延时[0000.15]
OUT 834.15  ; #4-1电池注氦阀关到位标志[0000.15]
LD TR0
AND 19.05  ; #4-2电池注氦阀开
TIMX(550) 1480 D23  ; 氦检相关无传感器阀开关到位延时设定, #4-2电池注氦阀开到位感应延时[0000.00]
LD TR0
ANDNOT 19.05  ; #4-2电池注氦阀开
TIMX(550) 1481 D23  ; 氦检相关无传感器阀开关到位延时设定, #4-2电池注氦阀关到位感应延时[0000.01]
LD TR0
AND T1480  ; #4-2电池注氦阀开到位感应延时[0000.00]
OUT 835.00  ; #4-2电池注氦阀开到位标志[0000.00]
LD TR0
AND T1481  ; #4-2电池注氦阀关到位感应延时[0000.01]
OUT 835.01  ; #4-2电池注氦阀关到位标志[0000.01]
LD TR0
AND 19.06  ; #4-1电池破真空阀开
TIMX(550) 1482 D23  ; 氦检相关无传感器阀开关到位延时设定, #4-1电池破真空阀开到位感应延时[0000.02]
LD TR0
ANDNOT 19.06  ; #4-1电池破真空阀开
TIMX(550) 1483 D23  ; 氦检相关无传感器阀开关到位延时设定, #4-1电池破真空阀关到位感应延时[0000.03]
LD TR0
AND T1482  ; #4-1电池破真空阀开到位感应延时[0000.02]
OUT 835.02  ; #4-1电池破真空阀开到位标志[0000.02]
LD TR0
AND T1483  ; #4-1电池破真空阀关到位感应延时[0000.03]
OUT 835.03  ; #4-1电池破真空阀关到位标志[0000.03]
LD TR0
AND 19.07  ; #4-2电池破真空阀开
TIMX(550) 1484 D23  ; 氦检相关无传感器阀开关到位延时设定, #4-2电池破真空阀开到位感应延时[0000.04]
LD TR0
ANDNOT 19.07  ; #4-2电池破真空阀开
TIMX(550) 1485 D23  ; 氦检相关无传感器阀开关到位延时设定, #4-2电池破真空阀关到位感应延时[0000.05]
LD TR0
AND T1484  ; #4-2电池破真空阀开到位感应延时[0000.04]
OUT 835.04  ; #4-2电池破真空阀开到位标志[0000.04]
LD TR0
AND T1485  ; #4-2电池破真空阀关到位感应延时[0000.05]
OUT 835.05  ; #4-2电池破真空阀关到位标志[0000.05]

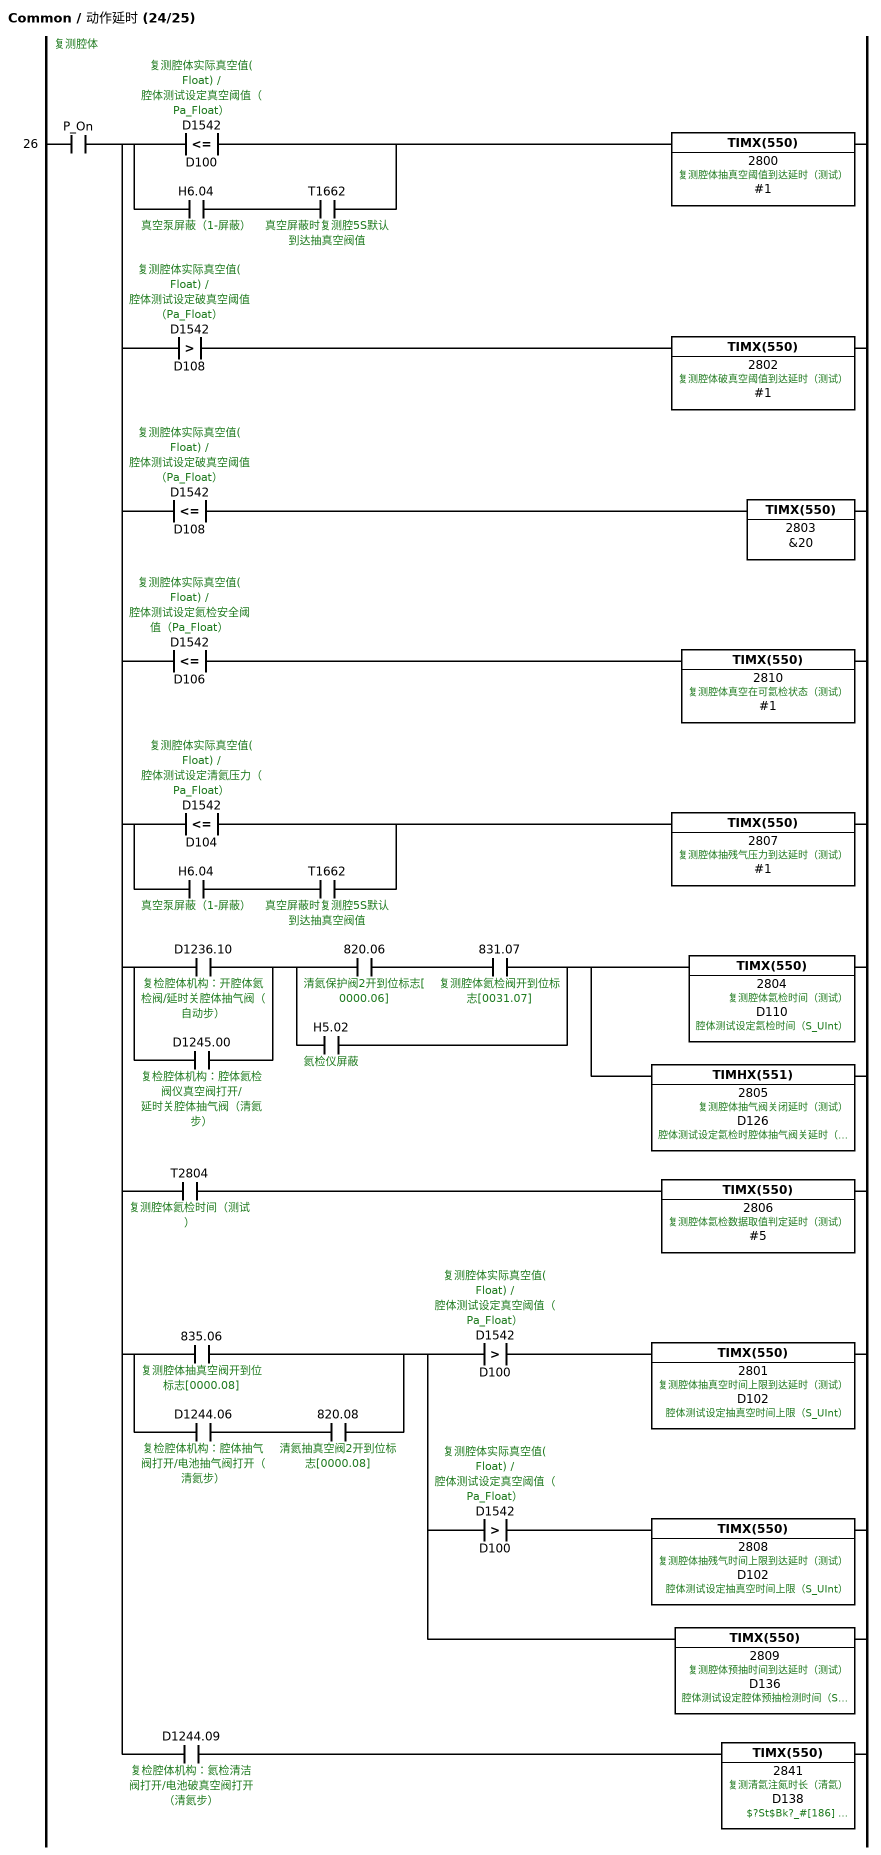
; rung 26: 复测腔体
LD P_On
OUT TR0
LD<=F(332) D1542 D100  ; 复测腔体实际真空值(Float), 腔体测试设定真空阈值（Pa_Float）
LD H6.04  ; 真空泵屏蔽（1-屏蔽）
AND T1662  ; 真空屏蔽时复测腔5S默认到达抽真空阀值
ORLD
ANDLD
TIMX(550) 2800 #1  ; 复测腔体抽真空阈值到达延时（测试）
LD TR0
AND>F(333) D1542 D108  ; 复测腔体实际真空值(Float), 腔体测试设定破真空阈值（Pa_Float）
TIMX(550) 2802 #1  ; 复测腔体破真空阈值到达延时（测试）
LD TR0
AND<=F(332) D1542 D108  ; 复测腔体实际真空值(Float), 腔体测试设定破真空阈值（Pa_Float）
TIMX(550) 2803 &20
LD TR0
AND<=F(332) D1542 D106  ; 复测腔体实际真空值(Float), 腔体测试设定氦检安全阈值（Pa_Float）
TIMX(550) 2810 #1  ; 复测腔体真空在可氦检状态（测试）
LD TR0
LD<=F(332) D1542 D104  ; 复测腔体实际真空值(Float), 腔体测试设定清氦压力（Pa_Float）
LD H6.04  ; 真空泵屏蔽（1-屏蔽）
AND T1662  ; 真空屏蔽时复测腔5S默认到达抽真空阀值
ORLD
ANDLD
TIMX(550) 2807 #1  ; 复测腔体抽残气压力到达延时（测试）
LD TR0
LD D1236.10  ; 复检腔体机构：开腔体氦检阀/延时关腔体抽气阀（自动步）
OR D1245.00  ; 复检腔体机构：腔体氦检阀仪真空阀打开/延时关腔体抽气阀（清氦步）
ANDLD
LD 820.06  ; 清氦保护阀2开到位标志[0000.06]
AND 831.07  ; 复测腔体氦检阀开到位标志[0031.07]
OR H5.02  ; 氦检仪屏蔽
ANDLD
TIMX(550) 2804 D110  ; 腔体测试设定氦检时间（S_UInt）, 复测腔体氦检时间（测试）
TIMHX(551) 2805 D126  ; 腔体测试设定氦检时腔体抽气阀关延时（S_UInt）, 复测腔体抽气阀关闭延时（测试）
LD TR0
AND T2804  ; 复测腔体氦检时间（测试）
TIMX(550) 2806 #5  ; 复测腔体氦检数据取值判定延时（测试）
LD TR0
LD 835.06  ; 复测腔体抽真空阀开到位标志[0000.08]
LD D1244.06  ; 复检腔体机构：腔体抽气阀打开/电池抽气阀打开（清氦步）
AND 820.08  ; 清氦抽真空阀2开到位标志[0000.08]
ORLD
ANDLD
OUT TR1
AND>F(333) D1542 D100  ; 复测腔体实际真空值(Float), 腔体测试设定真空阈值（Pa_Float）
TIMX(550) 2801 D102  ; 腔体测试设定抽真空时间上限（S_UInt）, 复测腔体抽真空时间上限到达延时（测试）
LD TR1
AND>F(333) D1542 D100  ; 复测腔体实际真空值(Float), 腔体测试设定真空阈值（Pa_Float）
TIMX(550) 2808 D102  ; 腔体测试设定抽真空时间上限（S_UInt）, 复测腔体抽残气时间上限到达延时（测试）
LD TR1
TIMX(550) 2809 D136  ; 腔体测试设定腔体预抽检测时间（S_UInt）, 复测腔体预抽时间到达延时（测试）
LD TR0
AND D1244.09  ; 复检腔体机构：氦检清洁阀打开/电池破真空阀打开（清氦步）
TIMX(550) 2841 D138  ; $?St$Bk?_#[186] / 管路清氦注氮时间（S_UInt） / $?St$Bk?_#[186], 复测清氦注氮时长（清氦）

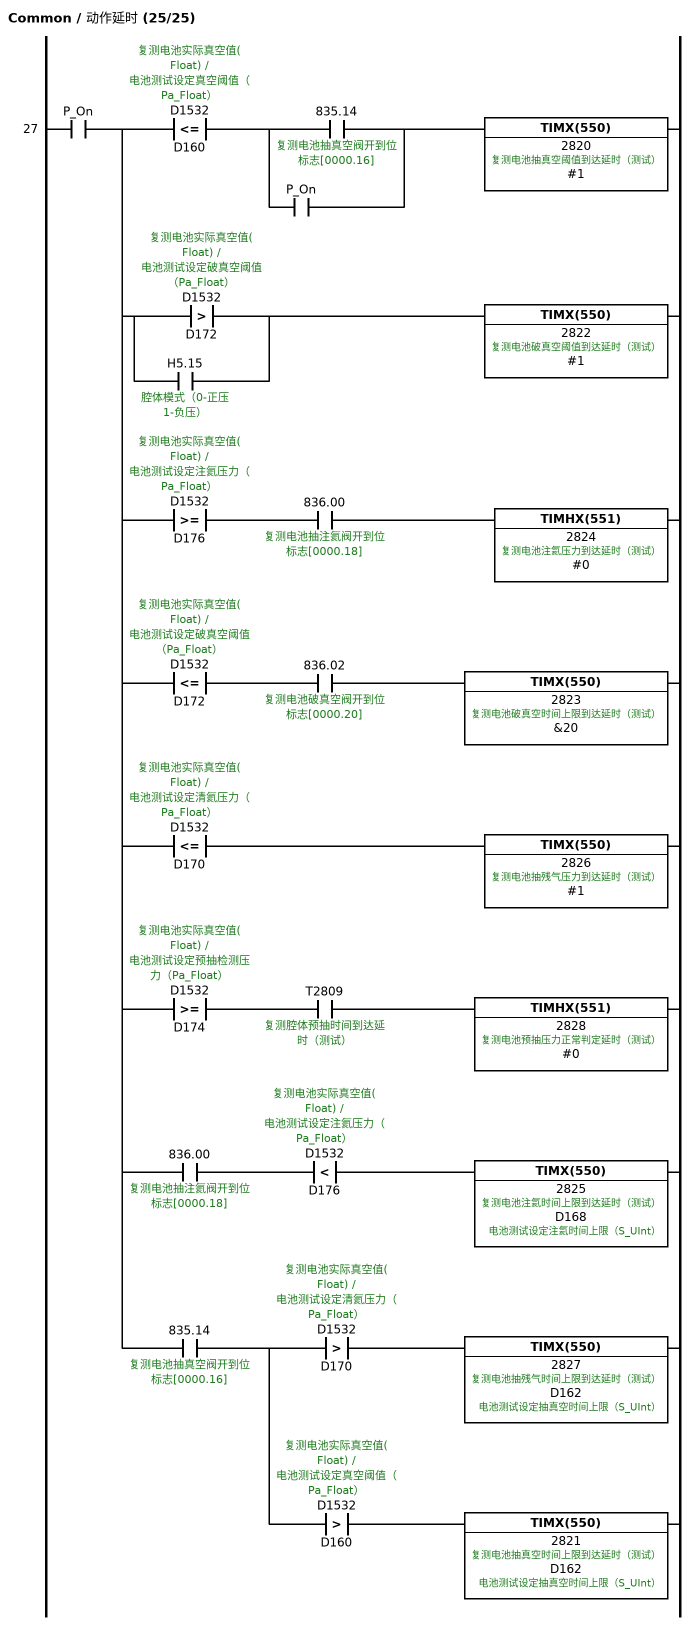
; rung 27
LD P_On
OUT TR0
AND<=F(332) D1532 D160  ; 复测电池实际真空值(Float), 电池测试设定真空阈值（Pa_Float）
LD 835.14  ; 复测电池抽真空阀开到位标志[0000.16]
OR P_On
ANDLD
TIMX(550) 2820 #1  ; 复测电池抽真空阈值到达延时（测试）
LD TR0
LD>F(333) D1532 D172  ; 复测电池实际真空值(Float), 电池测试设定破真空阈值（Pa_Float）
OR H5.15  ; 腔体模式（0-正压 1-负压）
ANDLD
TIMX(550) 2822 #1  ; 复测电池破真空阈值到达延时（测试）
LD TR0
AND>=F(334) D1532 D176  ; 复测电池实际真空值(Float), 电池测试设定注氦压力（Pa_Float）
AND 836.00  ; 复测电池抽注氦阀开到位标志[0000.18]
TIMHX(551) 2824 #0  ; 复测电池注氦压力到达延时（测试）
LD TR0
AND<=F(332) D1532 D172  ; 复测电池实际真空值(Float), 电池测试设定破真空阈值（Pa_Float）
AND 836.02  ; 复测电池破真空阀开到位标志[0000.20]
TIMX(550) 2823 &20  ; 复测电池破真空时间上限到达延时（测试）
LD TR0
AND<=F(332) D1532 D170  ; 复测电池实际真空值(Float), 电池测试设定清氦压力（Pa_Float）
TIMX(550) 2826 #1  ; 复测电池抽残气压力到达延时（测试）
LD TR0
AND>=F(334) D1532 D174  ; 复测电池实际真空值(Float), 电池测试设定预抽检测压力（Pa_Float）
AND T2809  ; 复测腔体预抽时间到达延时（测试）
TIMHX(551) 2828 #0  ; 复测电池预抽压力正常判定延时（测试）
LD TR0
AND 836.00  ; 复测电池抽注氦阀开到位标志[0000.18]
AND<F(331) D1532 D176  ; 复测电池实际真空值(Float), 电池测试设定注氦压力（Pa_Float）
TIMX(550) 2825 D168  ; 电池测试设定注氦时间上限（S_UInt）, 复测电池注氦时间上限到达延时（测试）
LD TR0
AND 835.14  ; 复测电池抽真空阀开到位标志[0000.16]
OUT TR0
AND>F(333) D1532 D170  ; 复测电池实际真空值(Float), 电池测试设定清氦压力（Pa_Float）
TIMX(550) 2827 D162  ; 电池测试设定抽真空时间上限（S_UInt）, 复测电池抽残气时间上限到达延时（测试）
LD TR0
AND>F(333) D1532 D160  ; 复测电池实际真空值(Float), 电池测试设定真空阈值（Pa_Float）
TIMX(550) 2821 D162  ; 电池测试设定抽真空时间上限（S_UInt）, 复测电池抽真空时间上限到达延时（测试）

### Section 传感器延时

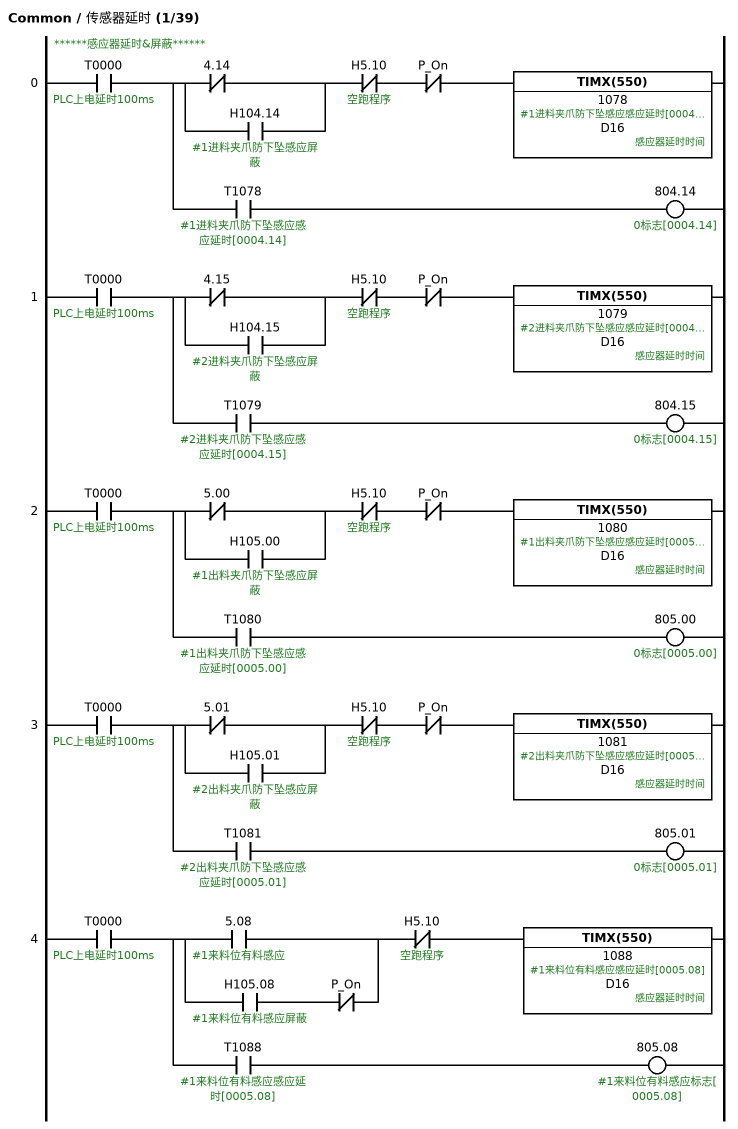
; rung 0: ******感应器延时&屏蔽******
LD T0000  ; PLC上电延时100ms
OUT TR0
LDNOT 4.14
OR H104.14  ; #1进料夹爪防下坠感应屏蔽
ANDLD
ANDNOT H5.10  ; 空跑程序
ANDNOT P_On
TIMX(550) 1078 D16  ; 感应器延时时间, #1进料夹爪防下坠感应感应延时[0004.14]
LD TR0
AND T1078  ; #1进料夹爪防下坠感应感应延时[0004.14]
OUT 804.14  ; 0标志[0004.14]
; rung 1
LD T0000  ; PLC上电延时100ms
OUT TR0
LDNOT 4.15
OR H104.15  ; #2进料夹爪防下坠感应屏蔽
ANDLD
ANDNOT H5.10  ; 空跑程序
ANDNOT P_On
TIMX(550) 1079 D16  ; 感应器延时时间, #2进料夹爪防下坠感应感应延时[0004.15]
LD TR0
AND T1079  ; #2进料夹爪防下坠感应感应延时[0004.15]
OUT 804.15  ; 0标志[0004.15]
; rung 2
LD T0000  ; PLC上电延时100ms
OUT TR0
LDNOT 5.00
OR H105.00  ; #1出料夹爪防下坠感应屏蔽
ANDLD
ANDNOT H5.10  ; 空跑程序
ANDNOT P_On
TIMX(550) 1080 D16  ; 感应器延时时间, #1出料夹爪防下坠感应感应延时[0005.00]
LD TR0
AND T1080  ; #1出料夹爪防下坠感应感应延时[0005.00]
OUT 805.00  ; 0标志[0005.00]
; rung 3
LD T0000  ; PLC上电延时100ms
OUT TR0
LDNOT 5.01
OR H105.01  ; #2出料夹爪防下坠感应屏蔽
ANDLD
ANDNOT H5.10  ; 空跑程序
ANDNOT P_On
TIMX(550) 1081 D16  ; 感应器延时时间, #2出料夹爪防下坠感应感应延时[0005.01]
LD TR0
AND T1081  ; #2出料夹爪防下坠感应感应延时[0005.01]
OUT 805.01  ; 0标志[0005.01]
; rung 4
LD T0000  ; PLC上电延时100ms
OUT TR0
LD 5.08  ; #1来料位有料感应
LD H105.08  ; #1来料位有料感应屏蔽
ANDNOT P_On
ORLD
ANDLD
ANDNOT H5.10  ; 空跑程序
TIMX(550) 1088 D16  ; 感应器延时时间, #1来料位有料感应感应延时[0005.08]
LD TR0
AND T1088  ; #1来料位有料感应感应延时[0005.08]
OUT 805.08  ; #1来料位有料感应标志[0005.08]

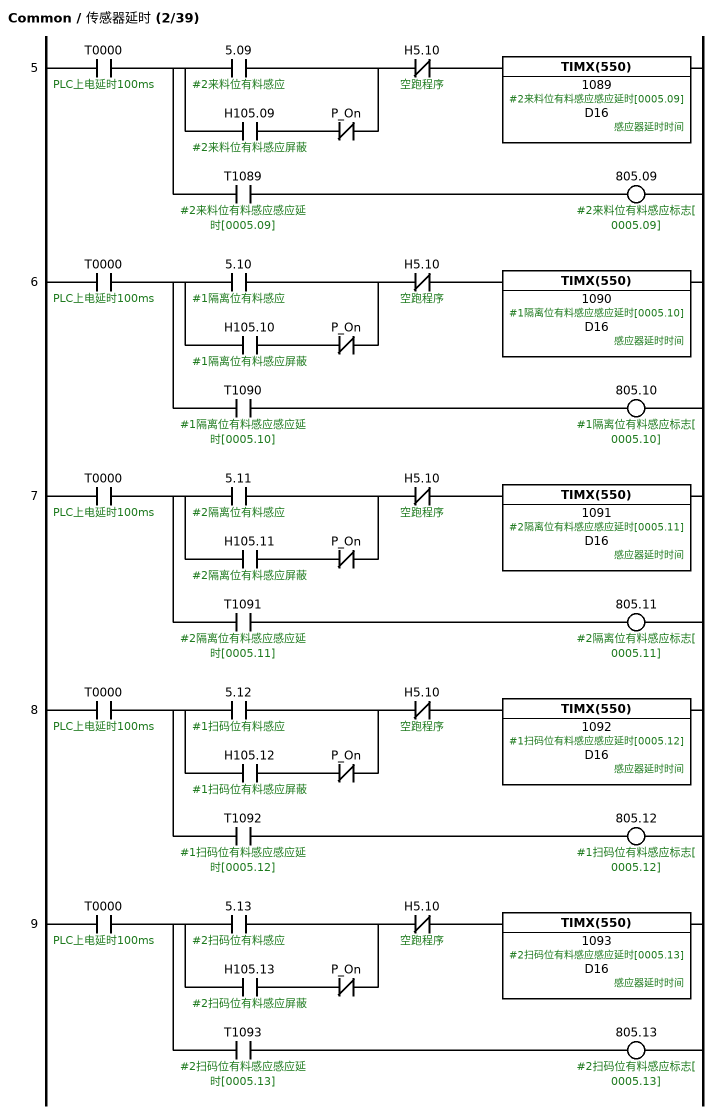
; rung 5
LD T0000  ; PLC上电延时100ms
OUT TR0
LD 5.09  ; #2来料位有料感应
LD H105.09  ; #2来料位有料感应屏蔽
ANDNOT P_On
ORLD
ANDLD
ANDNOT H5.10  ; 空跑程序
TIMX(550) 1089 D16  ; 感应器延时时间, #2来料位有料感应感应延时[0005.09]
LD TR0
AND T1089  ; #2来料位有料感应感应延时[0005.09]
OUT 805.09  ; #2来料位有料感应标志[0005.09]
; rung 6
LD T0000  ; PLC上电延时100ms
OUT TR0
LD 5.10  ; #1隔离位有料感应
LD H105.10  ; #1隔离位有料感应屏蔽
ANDNOT P_On
ORLD
ANDLD
ANDNOT H5.10  ; 空跑程序
TIMX(550) 1090 D16  ; 感应器延时时间, #1隔离位有料感应感应延时[0005.10]
LD TR0
AND T1090  ; #1隔离位有料感应感应延时[0005.10]
OUT 805.10  ; #1隔离位有料感应标志[0005.10]
; rung 7
LD T0000  ; PLC上电延时100ms
OUT TR0
LD 5.11  ; #2隔离位有料感应
LD H105.11  ; #2隔离位有料感应屏蔽
ANDNOT P_On
ORLD
ANDLD
ANDNOT H5.10  ; 空跑程序
TIMX(550) 1091 D16  ; 感应器延时时间, #2隔离位有料感应感应延时[0005.11]
LD TR0
AND T1091  ; #2隔离位有料感应感应延时[0005.11]
OUT 805.11  ; #2隔离位有料感应标志[0005.11]
; rung 8
LD T0000  ; PLC上电延时100ms
OUT TR0
LD 5.12  ; #1扫码位有料感应
LD H105.12  ; #1扫码位有料感应屏蔽
ANDNOT P_On
ORLD
ANDLD
ANDNOT H5.10  ; 空跑程序
TIMX(550) 1092 D16  ; 感应器延时时间, #1扫码位有料感应感应延时[0005.12]
LD TR0
AND T1092  ; #1扫码位有料感应感应延时[0005.12]
OUT 805.12  ; #1扫码位有料感应标志[0005.12]
; rung 9
LD T0000  ; PLC上电延时100ms
OUT TR0
LD 5.13  ; #2扫码位有料感应
LD H105.13  ; #2扫码位有料感应屏蔽
ANDNOT P_On
ORLD
ANDLD
ANDNOT H5.10  ; 空跑程序
TIMX(550) 1093 D16  ; 感应器延时时间, #2扫码位有料感应感应延时[0005.13]
LD TR0
AND T1093  ; #2扫码位有料感应感应延时[0005.13]
OUT 805.13  ; #2扫码位有料感应标志[0005.13]

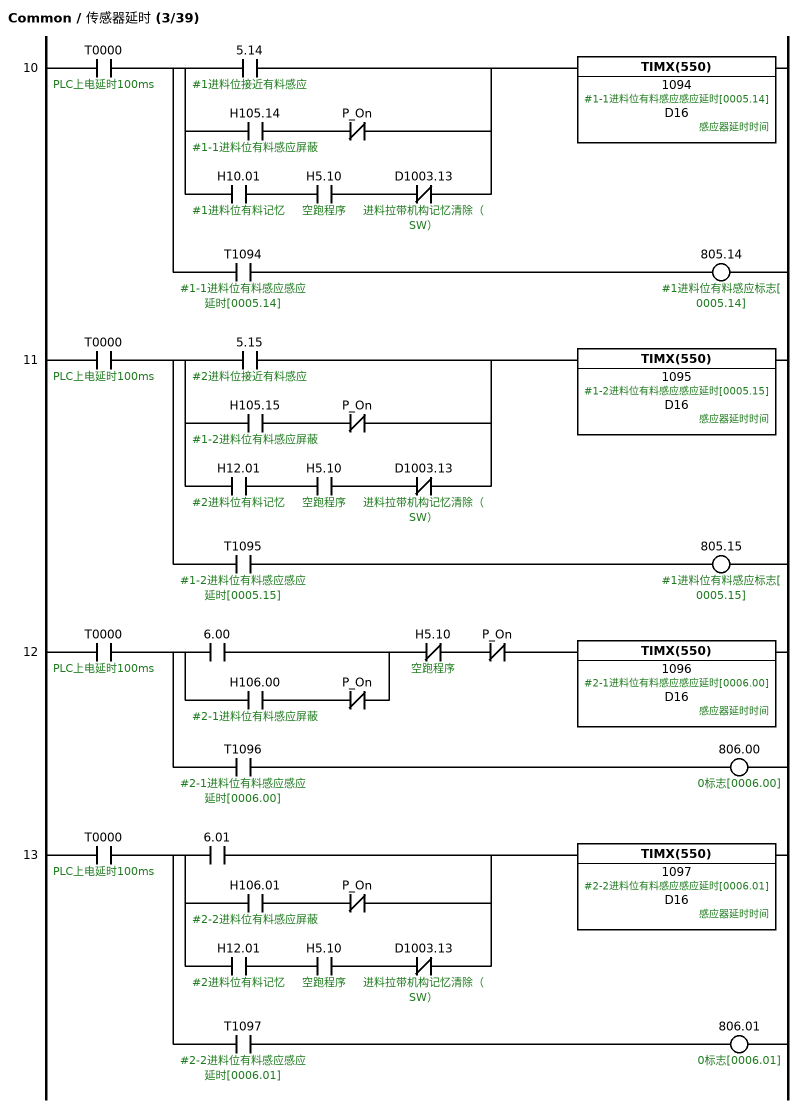
; rung 10
LD T0000  ; PLC上电延时100ms
OUT TR0
LD 5.14  ; #1进料位接近有料感应
LD H105.14  ; #1-1进料位有料感应屏蔽
ANDNOT P_On
ORLD
LD H10.01  ; #1进料位有料记忆
AND H5.10  ; 空跑程序
ANDNOT D1003.13  ; 进料拉带机构记忆清除（SW）
ORLD
ANDLD
TIMX(550) 1094 D16  ; 感应器延时时间, #1-1进料位有料感应感应延时[0005.14]
LD TR0
AND T1094  ; #1-1进料位有料感应感应延时[0005.14]
OUT 805.14  ; #1进料位有料感应标志[0005.14]
; rung 11
LD T0000  ; PLC上电延时100ms
OUT TR0
LD 5.15  ; #2进料位接近有料感应
LD H105.15  ; #1-2进料位有料感应屏蔽
ANDNOT P_On
ORLD
LD H12.01  ; #2进料位有料记忆
AND H5.10  ; 空跑程序
ANDNOT D1003.13  ; 进料拉带机构记忆清除（SW）
ORLD
ANDLD
TIMX(550) 1095 D16  ; 感应器延时时间, #1-2进料位有料感应感应延时[0005.15]
LD TR0
AND T1095  ; #1-2进料位有料感应感应延时[0005.15]
OUT 805.15  ; #1进料位有料感应标志[0005.15]
; rung 12
LD T0000  ; PLC上电延时100ms
OUT TR0
LD 6.00
LD H106.00  ; #2-1进料位有料感应屏蔽
ANDNOT P_On
ORLD
ANDLD
ANDNOT H5.10  ; 空跑程序
ANDNOT P_On
TIMX(550) 1096 D16  ; 感应器延时时间, #2-1进料位有料感应感应延时[0006.00]
LD TR0
AND T1096  ; #2-1进料位有料感应感应延时[0006.00]
OUT 806.00  ; 0标志[0006.00]
; rung 13
LD T0000  ; PLC上电延时100ms
OUT TR0
LD 6.01
LD H106.01  ; #2-2进料位有料感应屏蔽
ANDNOT P_On
ORLD
LD H12.01  ; #2进料位有料记忆
AND H5.10  ; 空跑程序
ANDNOT D1003.13  ; 进料拉带机构记忆清除（SW）
ORLD
ANDLD
TIMX(550) 1097 D16  ; 感应器延时时间, #2-2进料位有料感应感应延时[0006.01]
LD TR0
AND T1097  ; #2-2进料位有料感应感应延时[0006.01]
OUT 806.01  ; 0标志[0006.01]

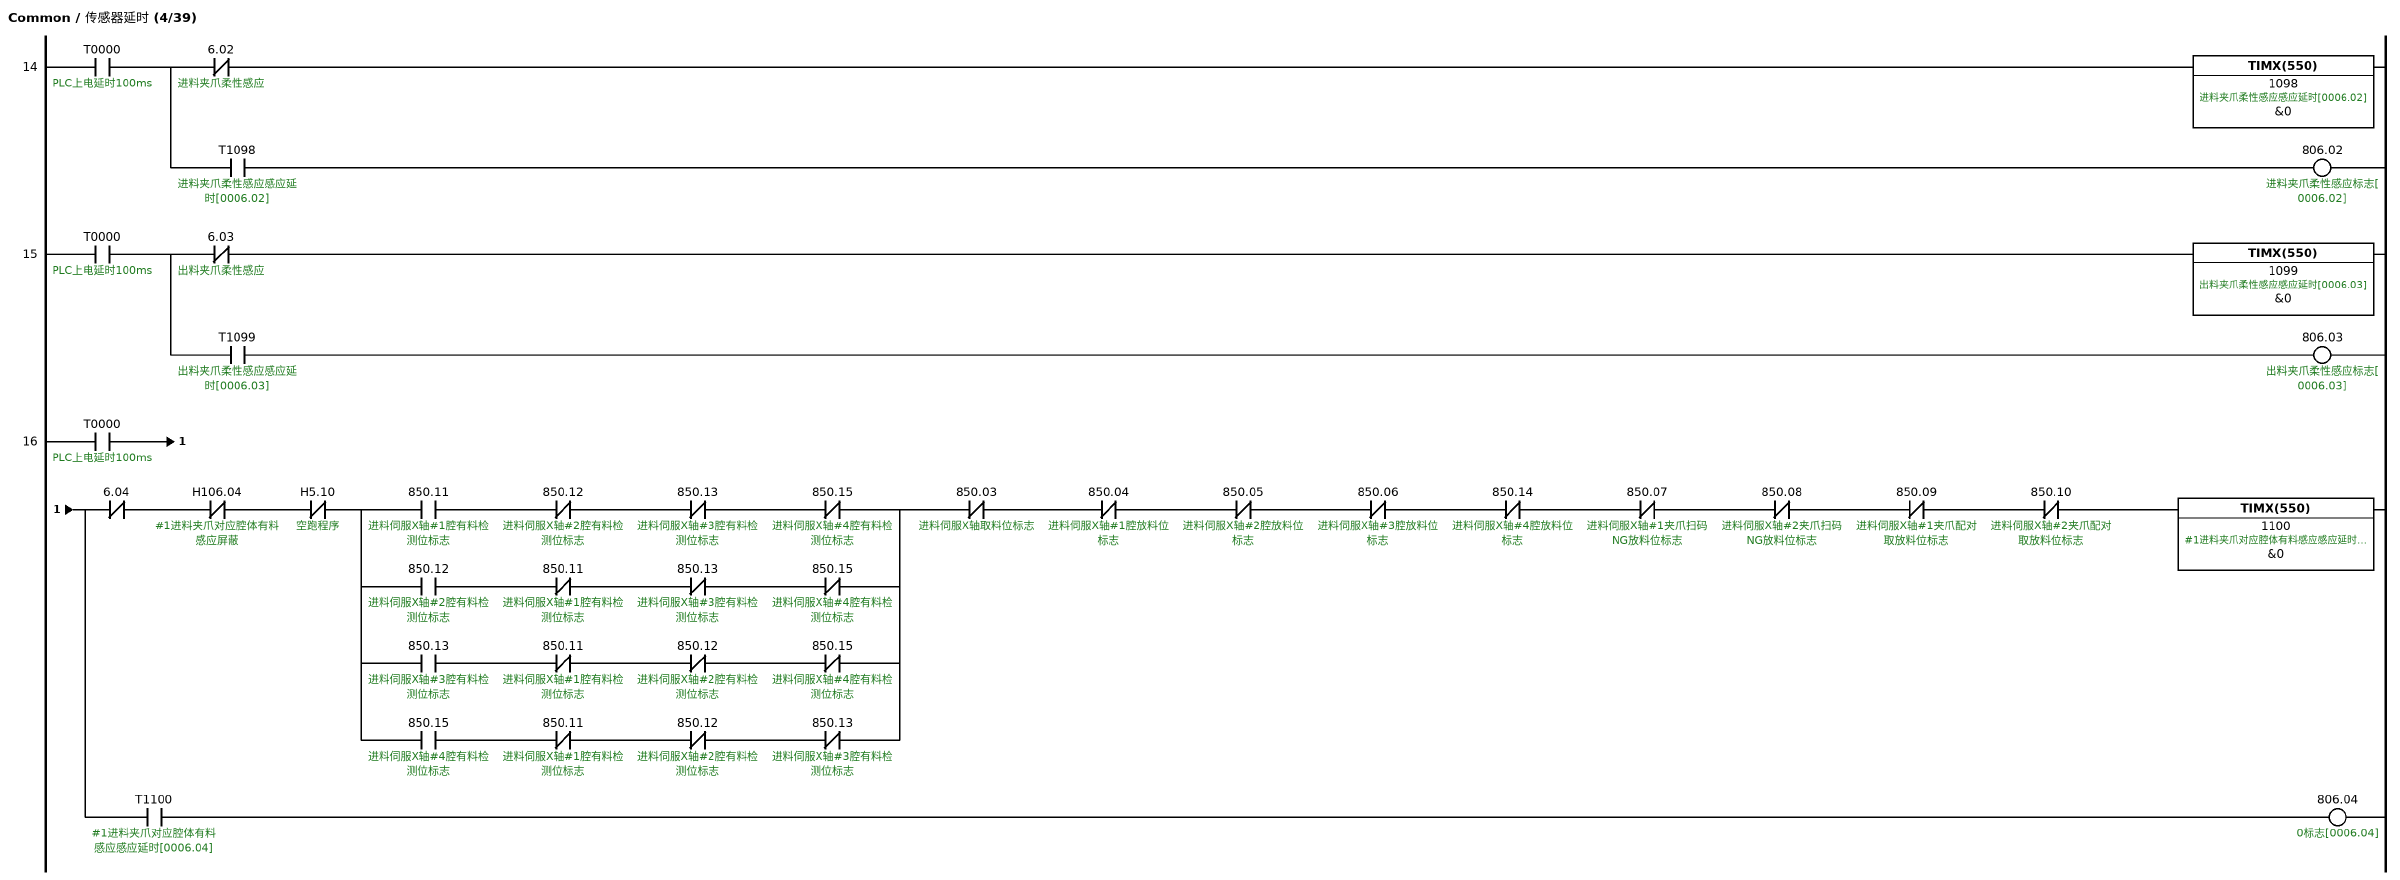
; rung 14
LD T0000  ; PLC上电延时100ms
OUT TR0
ANDNOT 6.02  ; 进料夹爪柔性感应
TIMX(550) 1098 &0  ; 进料夹爪柔性感应感应延时[0006.02]
LD TR0
AND T1098  ; 进料夹爪柔性感应感应延时[0006.02]
OUT 806.02  ; 进料夹爪柔性感应标志[0006.02]
; rung 15
LD T0000  ; PLC上电延时100ms
OUT TR0
ANDNOT 6.03  ; 出料夹爪柔性感应
TIMX(550) 1099 &0  ; 出料夹爪柔性感应感应延时[0006.03]
LD TR0
AND T1099  ; 出料夹爪柔性感应感应延时[0006.03]
OUT 806.03  ; 出料夹爪柔性感应标志[0006.03]
; rung 16
LD T0000  ; PLC上电延时100ms
OUT TR0
ANDNOT 6.04
ANDNOT H106.04  ; #1进料夹爪对应腔体有料感应屏蔽
ANDNOT H5.10  ; 空跑程序
LD 850.11  ; 进料伺服X轴#1腔有料检测位标志
ANDNOT 850.12  ; 进料伺服X轴#2腔有料检测位标志
ANDNOT 850.13  ; 进料伺服X轴#3腔有料检测位标志
ANDNOT 850.15  ; 进料伺服X轴#4腔有料检测位标志
LD 850.12  ; 进料伺服X轴#2腔有料检测位标志
ANDNOT 850.11  ; 进料伺服X轴#1腔有料检测位标志
ANDNOT 850.13  ; 进料伺服X轴#3腔有料检测位标志
ANDNOT 850.15  ; 进料伺服X轴#4腔有料检测位标志
ORLD
LD 850.13  ; 进料伺服X轴#3腔有料检测位标志
ANDNOT 850.11  ; 进料伺服X轴#1腔有料检测位标志
ANDNOT 850.12  ; 进料伺服X轴#2腔有料检测位标志
ANDNOT 850.15  ; 进料伺服X轴#4腔有料检测位标志
ORLD
LD 850.15  ; 进料伺服X轴#4腔有料检测位标志
ANDNOT 850.11  ; 进料伺服X轴#1腔有料检测位标志
ANDNOT 850.12  ; 进料伺服X轴#2腔有料检测位标志
ANDNOT 850.13  ; 进料伺服X轴#3腔有料检测位标志
ORLD
ANDLD
ANDNOT 850.03  ; 进料伺服X轴取料位标志
ANDNOT 850.04  ; 进料伺服X轴#1腔放料位标志
ANDNOT 850.05  ; 进料伺服X轴#2腔放料位标志
ANDNOT 850.06  ; 进料伺服X轴#3腔放料位标志
ANDNOT 850.14  ; 进料伺服X轴#4腔放料位标志
ANDNOT 850.07  ; 进料伺服X轴#1夹爪扫码NG放料位标志
ANDNOT 850.08  ; 进料伺服X轴#2夹爪扫码NG放料位标志
ANDNOT 850.09  ; 进料伺服X轴#1夹爪配对取放料位标志
ANDNOT 850.10  ; 进料伺服X轴#2夹爪配对取放料位标志
TIMX(550) 1100 &0  ; #1进料夹爪对应腔体有料感应感应延时[0006.04]
LD TR0
AND T1100  ; #1进料夹爪对应腔体有料感应感应延时[0006.04]
OUT 806.04  ; 0标志[0006.04]

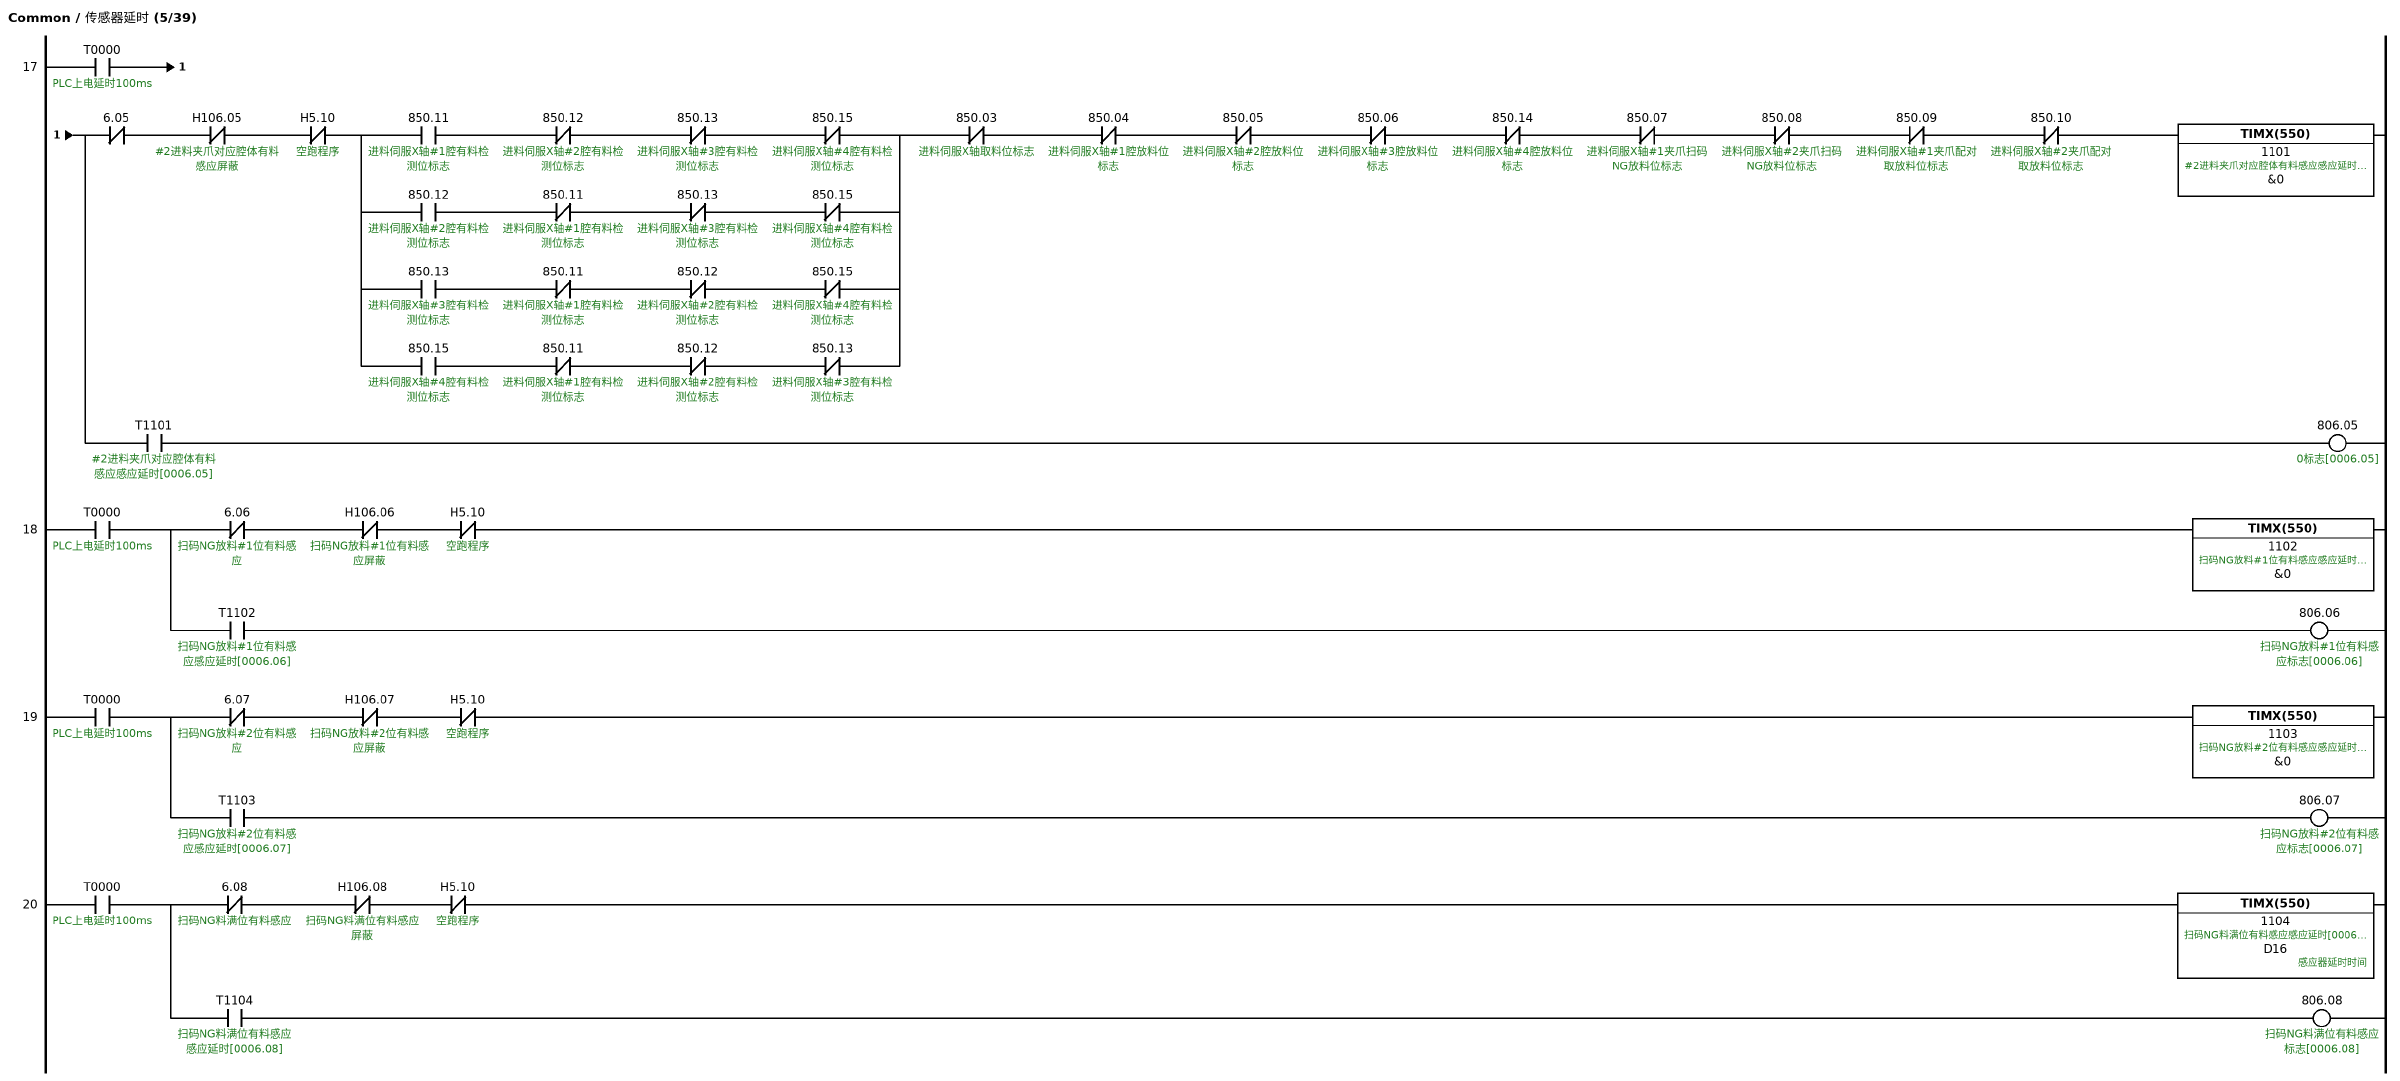
; rung 17
LD T0000  ; PLC上电延时100ms
OUT TR0
ANDNOT 6.05
ANDNOT H106.05  ; #2进料夹爪对应腔体有料感应屏蔽
ANDNOT H5.10  ; 空跑程序
LD 850.11  ; 进料伺服X轴#1腔有料检测位标志
ANDNOT 850.12  ; 进料伺服X轴#2腔有料检测位标志
ANDNOT 850.13  ; 进料伺服X轴#3腔有料检测位标志
ANDNOT 850.15  ; 进料伺服X轴#4腔有料检测位标志
LD 850.12  ; 进料伺服X轴#2腔有料检测位标志
ANDNOT 850.11  ; 进料伺服X轴#1腔有料检测位标志
ANDNOT 850.13  ; 进料伺服X轴#3腔有料检测位标志
ANDNOT 850.15  ; 进料伺服X轴#4腔有料检测位标志
ORLD
LD 850.13  ; 进料伺服X轴#3腔有料检测位标志
ANDNOT 850.11  ; 进料伺服X轴#1腔有料检测位标志
ANDNOT 850.12  ; 进料伺服X轴#2腔有料检测位标志
ANDNOT 850.15  ; 进料伺服X轴#4腔有料检测位标志
ORLD
LD 850.15  ; 进料伺服X轴#4腔有料检测位标志
ANDNOT 850.11  ; 进料伺服X轴#1腔有料检测位标志
ANDNOT 850.12  ; 进料伺服X轴#2腔有料检测位标志
ANDNOT 850.13  ; 进料伺服X轴#3腔有料检测位标志
ORLD
ANDLD
ANDNOT 850.03  ; 进料伺服X轴取料位标志
ANDNOT 850.04  ; 进料伺服X轴#1腔放料位标志
ANDNOT 850.05  ; 进料伺服X轴#2腔放料位标志
ANDNOT 850.06  ; 进料伺服X轴#3腔放料位标志
ANDNOT 850.14  ; 进料伺服X轴#4腔放料位标志
ANDNOT 850.07  ; 进料伺服X轴#1夹爪扫码NG放料位标志
ANDNOT 850.08  ; 进料伺服X轴#2夹爪扫码NG放料位标志
ANDNOT 850.09  ; 进料伺服X轴#1夹爪配对取放料位标志
ANDNOT 850.10  ; 进料伺服X轴#2夹爪配对取放料位标志
TIMX(550) 1101 &0  ; #2进料夹爪对应腔体有料感应感应延时[0006.05]
LD TR0
AND T1101  ; #2进料夹爪对应腔体有料感应感应延时[0006.05]
OUT 806.05  ; 0标志[0006.05]
; rung 18
LD T0000  ; PLC上电延时100ms
OUT TR0
ANDNOT 6.06  ; 扫码NG放料#1位有料感应
ANDNOT H106.06  ; 扫码NG放料#1位有料感应屏蔽
ANDNOT H5.10  ; 空跑程序
TIMX(550) 1102 &0  ; 扫码NG放料#1位有料感应感应延时[0006.06]
LD TR0
AND T1102  ; 扫码NG放料#1位有料感应感应延时[0006.06]
OUT 806.06  ; 扫码NG放料#1位有料感应标志[0006.06]
; rung 19
LD T0000  ; PLC上电延时100ms
OUT TR0
ANDNOT 6.07  ; 扫码NG放料#2位有料感应
ANDNOT H106.07  ; 扫码NG放料#2位有料感应屏蔽
ANDNOT H5.10  ; 空跑程序
TIMX(550) 1103 &0  ; 扫码NG放料#2位有料感应感应延时[0006.07]
LD TR0
AND T1103  ; 扫码NG放料#2位有料感应感应延时[0006.07]
OUT 806.07  ; 扫码NG放料#2位有料感应标志[0006.07]
; rung 20
LD T0000  ; PLC上电延时100ms
OUT TR0
ANDNOT 6.08  ; 扫码NG料满位有料感应
ANDNOT H106.08  ; 扫码NG料满位有料感应屏蔽
ANDNOT H5.10  ; 空跑程序
TIMX(550) 1104 D16  ; 感应器延时时间, 扫码NG料满位有料感应感应延时[0006.08]
LD TR0
AND T1104  ; 扫码NG料满位有料感应感应延时[0006.08]
OUT 806.08  ; 扫码NG料满位有料感应标志[0006.08]

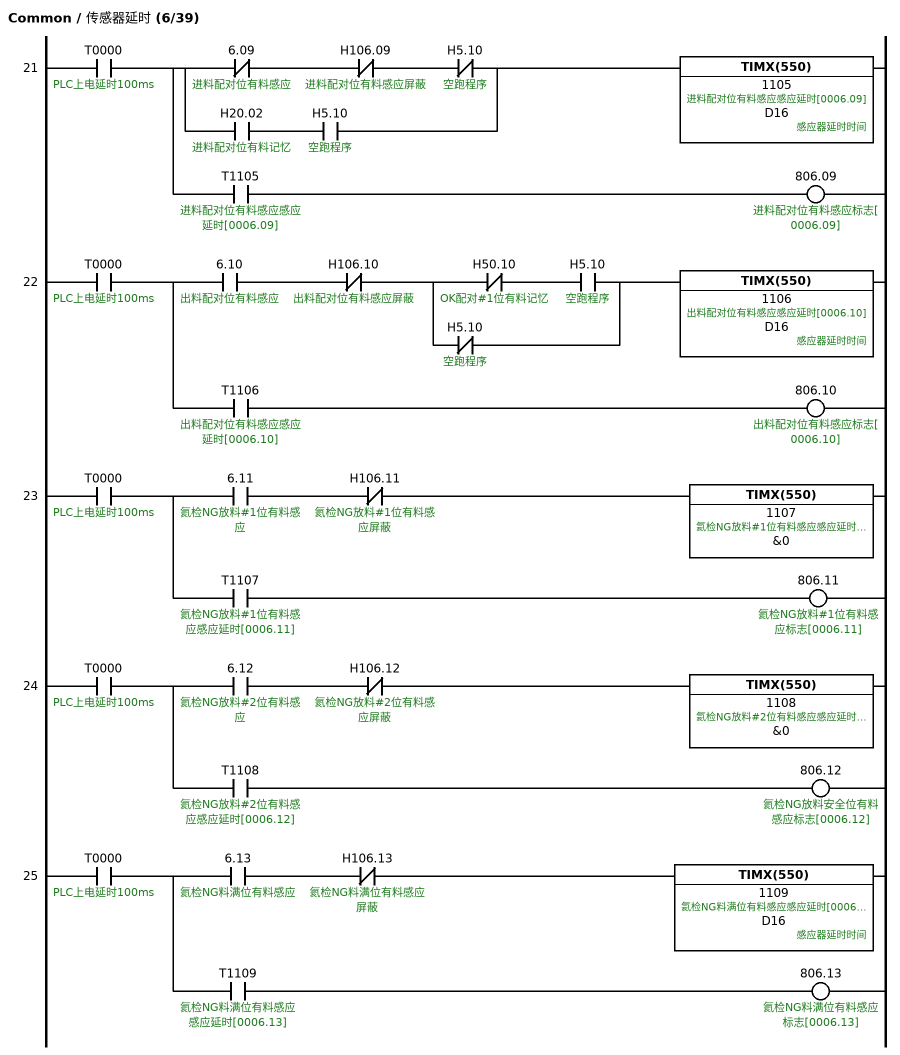
; rung 21
LD T0000  ; PLC上电延时100ms
OUT TR0
LDNOT 6.09  ; 进料配对位有料感应
ANDNOT H106.09  ; 进料配对位有料感应屏蔽
ANDNOT H5.10  ; 空跑程序
LD H20.02  ; 进料配对位有料记忆
AND H5.10  ; 空跑程序
ORLD
ANDLD
TIMX(550) 1105 D16  ; 感应器延时时间, 进料配对位有料感应感应延时[0006.09]
LD TR0
AND T1105  ; 进料配对位有料感应感应延时[0006.09]
OUT 806.09  ; 进料配对位有料感应标志[0006.09]
; rung 22
LD T0000  ; PLC上电延时100ms
OUT TR0
AND 6.10  ; 出料配对位有料感应
ANDNOT H106.10  ; 出料配对位有料感应屏蔽
LDNOT H50.10  ; OK配对#1位有料记忆
AND H5.10  ; 空跑程序
ORNOT H5.10  ; 空跑程序
ANDLD
TIMX(550) 1106 D16  ; 感应器延时时间, 出料配对位有料感应感应延时[0006.10]
LD TR0
AND T1106  ; 出料配对位有料感应感应延时[0006.10]
OUT 806.10  ; 出料配对位有料感应标志[0006.10]
; rung 23
LD T0000  ; PLC上电延时100ms
OUT TR0
AND 6.11  ; 氦检NG放料#1位有料感应
ANDNOT H106.11  ; 氦检NG放料#1位有料感应屏蔽
TIMX(550) 1107 &0  ; 氦检NG放料#1位有料感应感应延时[0006.11]
LD TR0
AND T1107  ; 氦检NG放料#1位有料感应感应延时[0006.11]
OUT 806.11  ; 氦检NG放料#1位有料感应标志[0006.11]
; rung 24
LD T0000  ; PLC上电延时100ms
OUT TR0
AND 6.12  ; 氦检NG放料#2位有料感应
ANDNOT H106.12  ; 氦检NG放料#2位有料感应屏蔽
TIMX(550) 1108 &0  ; 氦检NG放料#2位有料感应感应延时[0006.12]
LD TR0
AND T1108  ; 氦检NG放料#2位有料感应感应延时[0006.12]
OUT 806.12  ; 氦检NG放料安全位有料感应标志[0006.12]
; rung 25
LD T0000  ; PLC上电延时100ms
OUT TR0
AND 6.13  ; 氦检NG料满位有料感应
ANDNOT H106.13  ; 氦检NG料满位有料感应屏蔽
TIMX(550) 1109 D16  ; 感应器延时时间, 氦检NG料满位有料感应感应延时[0006.13]
LD TR0
AND T1109  ; 氦检NG料满位有料感应感应延时[0006.13]
OUT 806.13  ; 氦检NG料满位有料感应标志[0006.13]

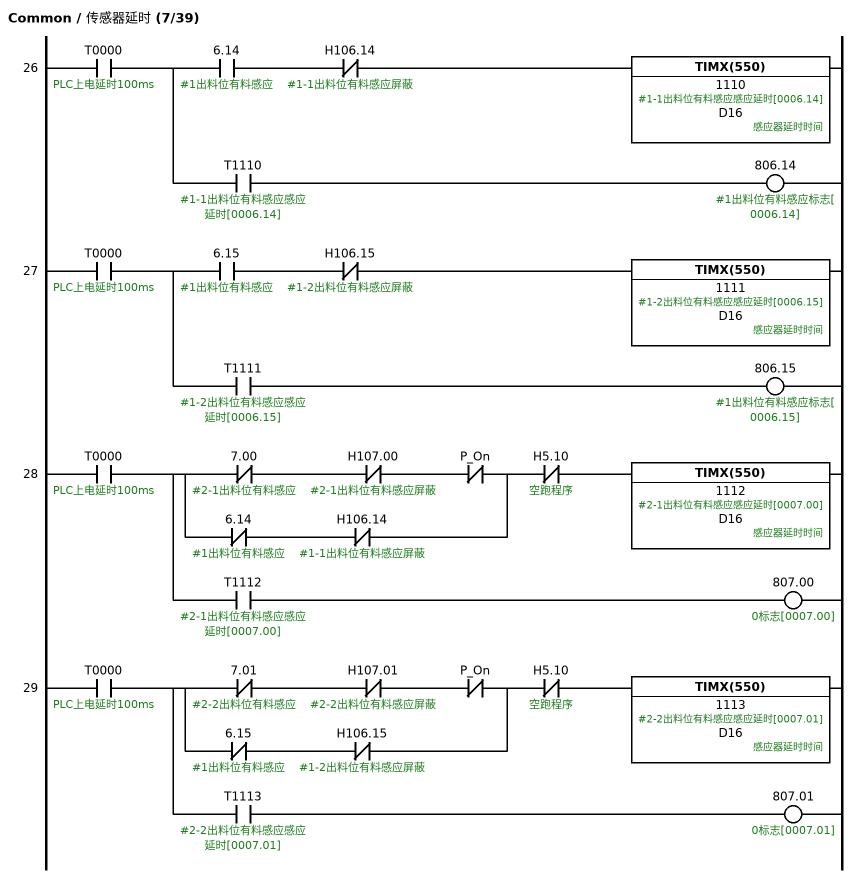
; rung 26
LD T0000  ; PLC上电延时100ms
OUT TR0
AND 6.14  ; #1出料位有料感应
ANDNOT H106.14  ; #1-1出料位有料感应屏蔽
TIMX(550) 1110 D16  ; 感应器延时时间, #1-1出料位有料感应感应延时[0006.14]
LD TR0
AND T1110  ; #1-1出料位有料感应感应延时[0006.14]
OUT 806.14  ; #1出料位有料感应标志[0006.14]
; rung 27
LD T0000  ; PLC上电延时100ms
OUT TR0
AND 6.15  ; #1出料位有料感应
ANDNOT H106.15  ; #1-2出料位有料感应屏蔽
TIMX(550) 1111 D16  ; 感应器延时时间, #1-2出料位有料感应感应延时[0006.15]
LD TR0
AND T1111  ; #1-2出料位有料感应感应延时[0006.15]
OUT 806.15  ; #1出料位有料感应标志[0006.15]
; rung 28
LD T0000  ; PLC上电延时100ms
OUT TR0
LDNOT 7.00  ; #2-1出料位有料感应
ANDNOT H107.00  ; #2-1出料位有料感应屏蔽
ANDNOT P_On
LDNOT 6.14  ; #1出料位有料感应
ANDNOT H106.14  ; #1-1出料位有料感应屏蔽
ORLD
ANDLD
ANDNOT H5.10  ; 空跑程序
TIMX(550) 1112 D16  ; 感应器延时时间, #2-1出料位有料感应感应延时[0007.00]
LD TR0
AND T1112  ; #2-1出料位有料感应感应延时[0007.00]
OUT 807.00  ; 0标志[0007.00]
; rung 29
LD T0000  ; PLC上电延时100ms
OUT TR0
LDNOT 7.01  ; #2-2出料位有料感应
ANDNOT H107.01  ; #2-2出料位有料感应屏蔽
ANDNOT P_On
LDNOT 6.15  ; #1出料位有料感应
ANDNOT H106.15  ; #1-2出料位有料感应屏蔽
ORLD
ANDLD
ANDNOT H5.10  ; 空跑程序
TIMX(550) 1113 D16  ; 感应器延时时间, #2-2出料位有料感应感应延时[0007.01]
LD TR0
AND T1113  ; #2-2出料位有料感应感应延时[0007.01]
OUT 807.01  ; 0标志[0007.01]

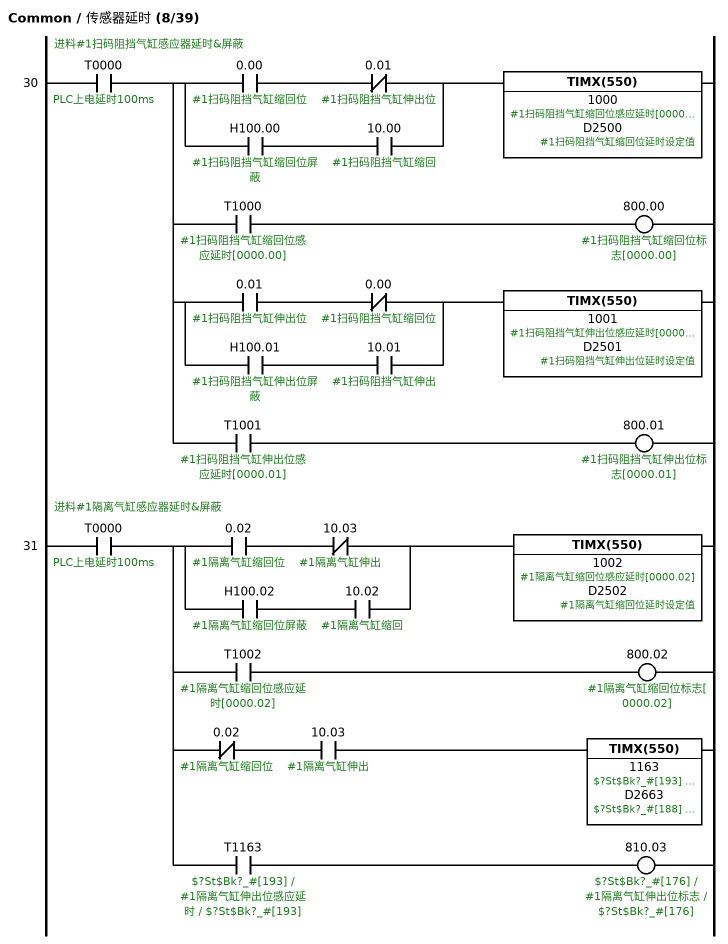
; rung 30: 进料#1扫码阻挡气缸感应器延时&屏蔽
LD T0000  ; PLC上电延时100ms
OUT TR0
LD 0.00  ; #1扫码阻挡气缸缩回位
ANDNOT 0.01  ; #1扫码阻挡气缸伸出位
LD H100.00  ; #1扫码阻挡气缸缩回位屏蔽
AND 10.00  ; #1扫码阻挡气缸缩回
ORLD
ANDLD
TIMX(550) 1000 D2500  ; #1扫码阻挡气缸缩回位延时设定值, #1扫码阻挡气缸缩回位感应延时[0000.00]
LD TR0
AND T1000  ; #1扫码阻挡气缸缩回位感应延时[0000.00]
OUT 800.00  ; #1扫码阻挡气缸缩回位标志[0000.00]
LD TR0
LD 0.01  ; #1扫码阻挡气缸伸出位
ANDNOT 0.00  ; #1扫码阻挡气缸缩回位
LD H100.01  ; #1扫码阻挡气缸伸出位屏蔽
AND 10.01  ; #1扫码阻挡气缸伸出
ORLD
ANDLD
TIMX(550) 1001 D2501  ; #1扫码阻挡气缸伸出位延时设定值, #1扫码阻挡气缸伸出位感应延时[0000.01]
LD TR0
AND T1001  ; #1扫码阻挡气缸伸出位感应延时[0000.01]
OUT 800.01  ; #1扫码阻挡气缸伸出位标志[0000.01]
; rung 31: 进料#1隔离气缸感应器延时&屏蔽
LD T0000  ; PLC上电延时100ms
OUT TR0
LD 0.02  ; #1隔离气缸缩回位
ANDNOT 10.03  ; #1隔离气缸伸出
LD H100.02  ; #1隔离气缸缩回位屏蔽
AND 10.02  ; #1隔离气缸缩回
ORLD
ANDLD
TIMX(550) 1002 D2502  ; #1隔离气缸缩回位延时设定值, #1隔离气缸缩回位感应延时[0000.02]
LD TR0
AND T1002  ; #1隔离气缸缩回位感应延时[0000.02]
OUT 800.02  ; #1隔离气缸缩回位标志[0000.02]
LD TR0
ANDNOT 0.02  ; #1隔离气缸缩回位
AND 10.03  ; #1隔离气缸伸出
TIMX(550) 1163 D2663  ; $?St$Bk?_#[188] / #1隔离气缸伸出位延时设定值 / $?St$Bk?_#[188], $?St$Bk?_#[193] / #1隔离气缸伸出位感应延时 / $?St$Bk?_#[193]
LD TR0
AND T1163  ; $?St$Bk?_#[193] / #1隔离气缸伸出位感应延时 / $?St$Bk?_#[193]
OUT 810.03  ; $?St$Bk?_#[176] / #1隔离气缸伸出位标志 / $?St$Bk?_#[176]

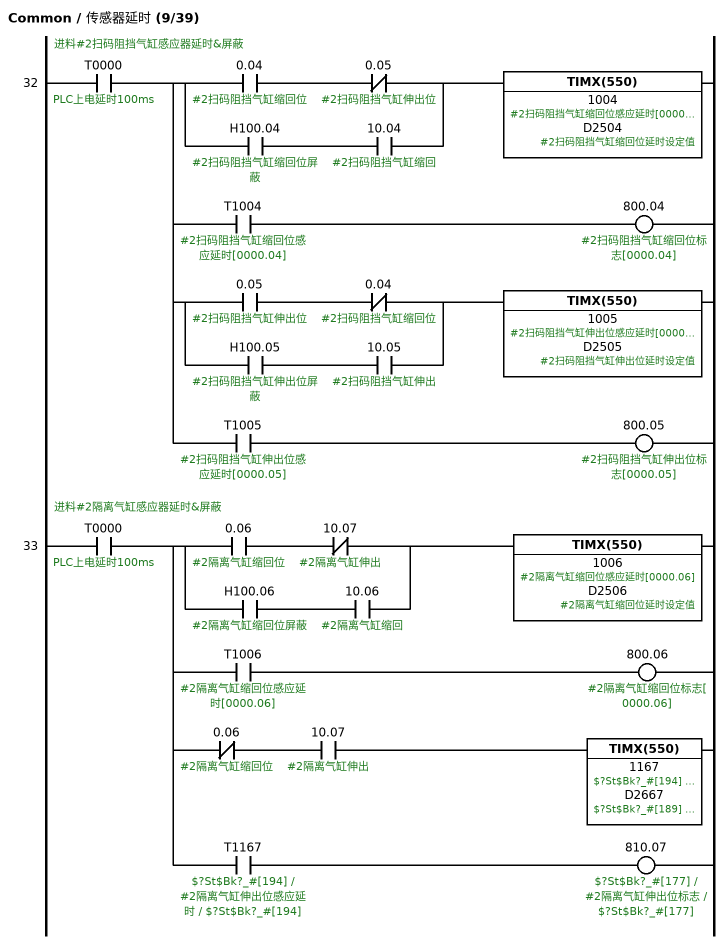
; rung 32: 进料#2扫码阻挡气缸感应器延时&屏蔽
LD T0000  ; PLC上电延时100ms
OUT TR0
LD 0.04  ; #2扫码阻挡气缸缩回位
ANDNOT 0.05  ; #2扫码阻挡气缸伸出位
LD H100.04  ; #2扫码阻挡气缸缩回位屏蔽
AND 10.04  ; #2扫码阻挡气缸缩回
ORLD
ANDLD
TIMX(550) 1004 D2504  ; #2扫码阻挡气缸缩回位延时设定值, #2扫码阻挡气缸缩回位感应延时[0000.04]
LD TR0
AND T1004  ; #2扫码阻挡气缸缩回位感应延时[0000.04]
OUT 800.04  ; #2扫码阻挡气缸缩回位标志[0000.04]
LD TR0
LD 0.05  ; #2扫码阻挡气缸伸出位
ANDNOT 0.04  ; #2扫码阻挡气缸缩回位
LD H100.05  ; #2扫码阻挡气缸伸出位屏蔽
AND 10.05  ; #2扫码阻挡气缸伸出
ORLD
ANDLD
TIMX(550) 1005 D2505  ; #2扫码阻挡气缸伸出位延时设定值, #2扫码阻挡气缸伸出位感应延时[0000.05]
LD TR0
AND T1005  ; #2扫码阻挡气缸伸出位感应延时[0000.05]
OUT 800.05  ; #2扫码阻挡气缸伸出位标志[0000.05]
; rung 33: 进料#2隔离气缸感应器延时&屏蔽
LD T0000  ; PLC上电延时100ms
OUT TR0
LD 0.06  ; #2隔离气缸缩回位
ANDNOT 10.07  ; #2隔离气缸伸出
LD H100.06  ; #2隔离气缸缩回位屏蔽
AND 10.06  ; #2隔离气缸缩回
ORLD
ANDLD
TIMX(550) 1006 D2506  ; #2隔离气缸缩回位延时设定值, #2隔离气缸缩回位感应延时[0000.06]
LD TR0
AND T1006  ; #2隔离气缸缩回位感应延时[0000.06]
OUT 800.06  ; #2隔离气缸缩回位标志[0000.06]
LD TR0
ANDNOT 0.06  ; #2隔离气缸缩回位
AND 10.07  ; #2隔离气缸伸出
TIMX(550) 1167 D2667  ; $?St$Bk?_#[189] / #2隔离气缸伸出位延时设定值 / $?St$Bk?_#[189], $?St$Bk?_#[194] / #2隔离气缸伸出位感应延时 / $?St$Bk?_#[194]
LD TR0
AND T1167  ; $?St$Bk?_#[194] / #2隔离气缸伸出位感应延时 / $?St$Bk?_#[194]
OUT 810.07  ; $?St$Bk?_#[177] / #2隔离气缸伸出位标志 / $?St$Bk?_#[177]

